					IF nCodingAndTrackingMode = 11 THEN
						FOR nPackIndex := 1 TO nMaxPackItem DO
							A_PackContentGenerator();
						END_FOR
					END_IF
	
					A_OuterEndPartGenerator();
					nOuterHeadCounter	:=nOuterHeadCounter +1;

				END_IF
	
			E_CS_ENDING:
				A_CaseEndPartGenerator();
				nCaseEndCounter :=	nCaseEndCounter	+1;
		END_CASE

		eState := E_XML_WRITEXML;
		nImigeProcessingSize	:= nImageByte;

	(* write XML file *)
	E_XML_WRITEXML:

		(* write XML image to file *)
		fbAppWriteFile(
			bExecute	:= TRUE,
			pSourceAddr	:= ADR(aXMLImage),
			nSourceSize	:= nImageByte,
			strPathFile	:= CONCAT(sPath, sFileName),
			tTimeout	:= T#3s,
		);

		(* file write complete *)
		IF fbAppWriteFile.bDone = TRUE THEN

			stWriteCHMFileStatistic.nTotalFilesWritten := stWriteCHMFileStatistic.nTotalFilesWritten + 1;

			(* file write completed OK *)
			IF fbAppWriteFile.bError = FALSE THEN

				(* correct no of bytes written to file *)
				IF fbAppWriteFile.nBytesWritten = nImageByte THEN

					stWriteCHMFileStatistic.nGoodFilesWritten := stWriteCHMFileStatistic.nGoodFilesWritten + 1;

					IF bCheckFileSize THEN
						eState := E_XML_CHECKFILESIZE;
					ELSE
						eState := E_XML_DONE;
					END_IF

				(* incorrect no of bytes written to file *)
				ELSE
					stWriteCHMFileStatistic.nBadFilesWritten :=stWriteCHMFileStatistic. nBadFilesWritten + 1;
				END_IF

			(* file write error *)
			ELSE

				bError := TRUE;
				nErrorID := fbAppWriteFile.nErrorID;
				eErrorState := eState;
				stWriteCHMFileStatistic.nFileWriteErrors := stWriteCHMFileStatistic.nFileWriteErrors + 1;

				eState := E_XML_DONE;
			END_IF

			(* close of fbWriteFile *)
			fbAppWriteFile(bExecute := FALSE);
		END_IF


	(* check XML file size is correct *)
	E_XML_CHECKFILESIZE:

		(* read XML file attributes *)
		fbGetFileInfo(
			bExecute		:= TRUE,
			strPathSource	:= sPath,
			strFileName	:= sFileName,
			tTimeout		:= T#1s,
		);

		(* read file attributes complete *)
		IF fbGetFileInfo.bDone = TRUE THEN

			stWriteCHMFileStatistic.nTotalFilesVerified := stWriteCHMFileStatistic.nTotalFilesVerified + 1;

			(* read file attributes completed OK *)
			IF fbGetFileInfo.bError = FALSE THEN

				(* file exists and file size is correct *)
				IF fbGetFileInfo.bFileExists = TRUE THEN

					(* file size is 0 bytes *)
					IF fbGetFileInfo.nFileSizeLo = 0 THEN

						stWriteCHMFileStatistic.nEmptyFilesVerified := stWriteCHMFileStatistic.nEmptyFilesVerified + 1;

					(* file size is not expected size *)
					ELSIF fbGetFileInfo.nFileSizeLo <> nImageByte THEN

						stWriteCHMFileStatistic.nSizeErrorsVerified :=stWriteCHMFileStatistic. nSizeErrorsVerified + 1;

					(* file size is correct *)
					ELSE

						stWriteCHMFileStatistic.nGoodFilesVerified := stWriteCHMFileStatistic.nGoodFilesVerified + 1;
					END_IF

					eState := E_XML_DONE;

				(* file not found *)
				ELSE

					bVerifyError := TRUE;
					stWriteCHMFileStatistic.nFileVerifyNotFound :=stWriteCHMFileStatistic.nFileVerifyNotFound + 1;

					IF bError = FALSE THEN

						bError := TRUE;
						nErrorID := 999;
						eErrorState := eState;
					END_IF

					eState := E_XML_DONE;
				END_IF

			(* read file attributes error *)
			ELSE

				stWriteCHMFileStatistic.nFileVerifyErrors := stWriteCHMFileStatistic.nFileVerifyErrors + 1;

				IF bError = FALSE THEN

					bError := TRUE;
					nErrorID := fbGetFileInfo.nErrorID;
					eErrorState := eState;
				END_IF

				eState := E_XML_DONE;
			END_IF

			(* close off fbFileSize *)
			fbGetFileInfo(bExecute := FALSE);
		END_IF


	(* sequence complete *)
	E_XML_DONE:

		(* update outputs *)
		bBusy := FALSE;
		bDone := TRUE;

		eState := E_XML_IDLE;
END_CASE

ACTION A_CaseEndPartGenerator:
	IF nCodingAndTrackingMode >= 7 THEN


				(* ItemList end*)
				sString := '$T$T$T$T</ItemList>$R$N';
				MEMMOVE(ADR(aXMLImage[nImageByte]), ADR(sString), LEN(sString));
				nImageByte := nImageByte + LEN(sString);

(***********CASE CONTENT END***********)
			(* Case Content END *)
			sString := '$T$T$T</Content>$R$N';
			MEMMOVE(ADR(aXMLImage[nImageByte]), ADR(sString), LEN(sString));
			nImageByte := nImageByte + LEN(sString);

	END_IF
			(* ProductionOrder *)
			sString := F_CONCAT3('$T$T$T<ProductionOrder>',stAgregationData.GenericHierarchy.CaseItem.ProductionOrder, '</ProductionOrder>$R$N');
			MEMMOVE(ADR(aXMLImage[nImageByte]), ADR(sString), LEN(sString));
			nImageByte := nImageByte + LEN(sString);

			(* LocalProductionOrder *)
			sString := F_CONCAT3('$T$T$T<LocalProductionOrder>',stAgregationData.GenericHierarchy.CaseItem.LocalProductionOrder, '</LocalProductionOrder>$R$N');
			MEMMOVE(ADR(aXMLImage[nImageByte]), ADR(sString), LEN(sString));
			nImageByte := nImageByte + LEN(sString);

			(* PITCode *)
			sString := F_CONCAT3('$T$T$T<PITCode>',stAgregationData.GenericHierarchy.CaseItem.PITCode, '</PITCode>$R$N');
			MEMMOVE(ADR(aXMLImage[nImageByte]), ADR(sString), LEN(sString));
			nImageByte := nImageByte + LEN(sString);

			(* BatchID *)
			sString := F_CONCAT3('$T$T$T<BatchID>',stAgregationData.GenericHierarchy.CaseItem.BatchID, '</BatchID>$R$N');
			MEMMOVE(ADR(aXMLImage[nImageByte]), ADR(sString), LEN(sString));
			nImageByte := nImageByte + LEN(sString);

			(* ProductionLine *)
			sString := F_CONCAT3('$T$T$T<ProductionLine>',stAgregationData.GenericHierarchy.CaseItem.ProductionLine, '</ProductionLine>$R$N');
			MEMMOVE(ADR(aXMLImage[nImageByte]), ADR(sString), LEN(sString));
			nImageByte := nImageByte + LEN(sString);


(***********Item CONTENT END***********)
		(* Item END *)
		sString := '$T$T</Item>$R$N';
		MEMMOVE(ADR(aXMLImage[nImageByte]), ADR(sString), LEN(sString));
		nImageByte := nImageByte + LEN(sString);

(***********GENERIC HIERARCHY CONTENT END***********)

	(* GenericHierarchy END *)
	sString := '$T</GenericHierarchy>$R$N';
	MEMMOVE(ADR(aXMLImage[nImageByte]), ADR(sString), LEN(sString));
	nImageByte := nImageByte + LEN(sString);

	(* Attributes *)
	sString := F_CONCAT3('$T<Attributes>', stAgregationData.Attributes.CSProductionTime, '</Attributes>$R$N');
	MEMMOVE(ADR(aXMLImage[nImageByte]), ADR(sString), LEN(sString));
	nImageByte := nImageByte + LEN(sString);

(* XPath leading tag  END*)
sString := '</GenericHierarchyList> $R$N';
MEMMOVE(ADR(aXMLImage[nImageByte]), ADR(sString), LEN(sString));
nImageByte := nImageByte + LEN(sString);
END_ACTION

ACTION A_CaseHeaderGenerator:
(* XML file version *)
(*sString := '<?xml version="1.0" encoding="utf-8"?>$R$N';
MEMMOVE(ADR(aXMLImage[nImageByte]), ADR(sString), LEN(sString));
nImageByte := nImageByte + LEN(sString);*)

(* XPath leading tag *)
sString := '<GenericHierarchyList xmlns:xsd="http://www.w3.org/2001/XMLSchema" xmlns:xsi="http://www.w3.org/2001/XMLSchema-instance"> $R$N';
MEMMOVE(ADR(aXMLImage[nImageByte]), ADR(sString), LEN(sString));
nImageByte := nImageByte + LEN(sString);

	(* MessageHeader *)
	sString := '$T<MessageHeader>$R$N';
	MEMMOVE(ADR(aXMLImage[nImageByte]), ADR(sString), LEN(sString));
	nImageByte := nImageByte + LEN(sString);

(***********MESSAGE HEADER CONTENT***********)

		(*(* CreationDate *)
		sString := F_CONCAT3('$T$T<CreationDate>',stAgregationData.MessageHeader.CreationDate, '</CreationDate>$R$N');
		MEMMOVE(ADR(aXMLImage[nImageByte]), ADR(sString), LEN(sString));
		nImageByte := nImageByte + LEN(sString);
	
		(* CreationTime *)
		sString := F_CONCAT3('$T$T<CreationTime>',stAgregationData.MessageHeader.CreationTime, '</CreationTime>$R$N');
		MEMMOVE(ADR(aXMLImage[nImageByte]), ADR(sString), LEN(sString));
		nImageByte := nImageByte + LEN(sString);*)

		(* ReferenceID *)
		sString := F_CONCAT3('$T$T<ReferenceID>',stAgregationData.MessageHeader.ReferenceID, '</ReferenceID>$R$N');
		MEMMOVE(ADR(aXMLImage[nImageByte]), ADR(sString), LEN(sString));
		nImageByte := nImageByte + LEN(sString);

		(* CreationTimeLocalUTC *)
		sString := F_CONCAT3('$T$T<CreationTimeLocalUTC>',stAgregationData.MessageHeader.CreationTimeLocalUTC, '</CreationTimeLocalUTC>$R$N');
		MEMMOVE(ADR(aXMLImage[nImageByte]), ADR(sString), LEN(sString));
		nImageByte := nImageByte + LEN(sString);

		(* MessageType *)
		sString := F_CONCAT3('$T$T<MessageType>',stAgregationData.MessageHeader.MessageType, '</MessageType>$R$N');
		MEMMOVE(ADR(aXMLImage[nImageByte]), ADR(sString), LEN(sString));
		nImageByte := nImageByte + LEN(sString);

		(* SenderSystem *)
		sString := F_CONCAT3('$T$T<SenderSystem>',stAgregationData.MessageHeader.SenderSystem, '</SenderSystem>$R$N');
		MEMMOVE(ADR(aXMLImage[nImageByte]), ADR(sString), LEN(sString));
		nImageByte := nImageByte + LEN(sString);

		(* ReceiverSystem *)
		sString := F_CONCAT3('$T$T<ReceiverSystem>',stAgregationData.MessageHeader.ReceiverSystem, '</ReceiverSystem>$R$N');
		MEMMOVE(ADR(aXMLImage[nImageByte]), ADR(sString), LEN(sString));
		nImageByte := nImageByte + LEN(sString);

(***********MESSAGE HEADER CONTENT END***********)

	(* MessageHeader END *)
	sString := '$T</MessageHeader>$R$N';
	MEMMOVE(ADR(aXMLImage[nImageByte]), ADR(sString), LEN(sString));
	nImageByte := nImageByte + LEN(sString);

	(* Factory*)
	sString := F_CONCAT3('$T<Factory>', stAgregationData.Factory, '</Factory>$R$N');
	MEMMOVE(ADR(aXMLImage[nImageByte]), ADR(sString), LEN(sString));
	nImageByte := nImageByte + LEN(sString);

	(* GenericHierarchy *)
	sString := '$T<GenericHierarchy>$R$N';
	MEMMOVE(ADR(aXMLImage[nImageByte]), ADR(sString), LEN(sString));
	nImageByte := nImageByte + LEN(sString);

(***********GENERIC HIERARCHY CONTENT***********)

		(* HierarchyType *)
		sString := F_CONCAT3('$T$T<HierarchyType>',stAgregationData.GenericHierarchy.HierarchyType, '</HierarchyType>$R$N');
		MEMMOVE(ADR(aXMLImage[nImageByte]), ADR(sString), LEN(sString));
		nImageByte := nImageByte + LEN(sString);

		(* PerformedAction *)
		sString := F_CONCAT3('$T$T<ACTION>',stAgregationData.GenericHierarchy.PerformedAction, '</ACTION>$R$N');
		MEMMOVE(ADR(aXMLImage[nImageByte]), ADR(sString), LEN(sString));
		nImageByte := nImageByte + LEN(sString);

		(* TrackingLevels *)
		sString := F_CONCAT3('$T$T<TrackingLevels>',stAgregationData.GenericHierarchy.TrackingLevels, '</TrackingLevels>$R$N');
		MEMMOVE(ADR(aXMLImage[nImageByte]), ADR(sString), LEN(sString));
		nImageByte := nImageByte + LEN(sString);

		(* TrackingIndicator *)
		sString := F_CONCAT3('$T$T<TrackingIndicator>',stAgregationData.GenericHierarchy.TrackingIndicator, '</TrackingIndicator>$R$N');
		MEMMOVE(ADR(aXMLImage[nImageByte]), ADR(sString), LEN(sString));
		nImageByte := nImageByte + LEN(sString);

		(* Item Type *)
		sString := '$T$T<Item Type="CS">$R$N';
		MEMMOVE(ADR(aXMLImage[nImageByte]), ADR(sString), LEN(sString));
		nImageByte := nImageByte + LEN(sString);

(***********Item Type CONTENT***********)
			(* Identity*)
			sString := '$T$T$T<Identity>$R$N';
			MEMMOVE(ADR(aXMLImage[nImageByte]), ADR(sString), LEN(sString));
			nImageByte := nImageByte + LEN(sString);

(***********Identity CONTENT***********)
					(* SKU *)
					sString := F_CONCAT3('$T$T$T$T<SKU>',stAgregationData.GenericHierarchy.CaseItem.Identity.SKU, '</SKU>$R$N');
					MEMMOVE(ADR(aXMLImage[nImageByte]), ADR(sString), LEN(sString));
					nImageByte := nImageByte + LEN(sString);

					(* GTIN *)
					sString := F_CONCAT3('$T$T$T$T<GTIN>',stAgregationData.GenericHierarchy.CaseItem.Identity.GTIN, '</GTIN>$R$N');
					MEMMOVE(ADR(aXMLImage[nImageByte]), ADR(sString), LEN(sString));
					nImageByte := nImageByte + LEN(sString);

					(* ID *)
					sString := F_CONCAT3('$T$T$T$T<ID>',stAgregationData.GenericHierarchy.CaseItem.Identity.ID, '</ID>$R$N');
					MEMMOVE(ADR(aXMLImage[nImageByte]), ADR(sString), LEN(sString));
					nImageByte := nImageByte + LEN(sString);

					(* ReadQuality *)
					sString := F_CONCAT3('$T$T$T$T<ReadQuality>',stAgregationData.GenericHierarchy.CaseItem.Identity.ReadQuality, '</ReadQuality>$R$N');
					MEMMOVE(ADR(aXMLImage[nImageByte]), ADR(sString), LEN(sString));
					nImageByte := nImageByte + LEN(sString);

(***********Identity CONTENT END***********)

			(* Identity END *)
			sString := '$T$T$T</Identity>$R$N';
			MEMMOVE(ADR(aXMLImage[nImageByte]), ADR(sString), LEN(sString));
			nImageByte := nImageByte + LEN(sString);

			(* ItemState *)
			sString := F_CONCAT3('$T$T$T<ItemState>',stAgregationData.GenericHierarchy.CaseItem.ItemState, '</ItemState>$R$N');
			MEMMOVE(ADR(aXMLImage[nImageByte]), ADR(sString), LEN(sString));
			nImageByte := nImageByte + LEN(sString);

			(* RejectReason *)
			sString := '$T$T$T<RejectReason>$R$N';
			MEMMOVE(ADR(aXMLImage[nImageByte]), ADR(sString), LEN(sString));
			nImageByte := nImageByte + LEN(sString);

				sString := F_CONCAT3('$T$T$T$T<Reason>',stAgregationData.GenericHierarchy.CaseItem.RejectReason, '</Reason>$R$N');
				MEMMOVE(ADR(aXMLImage[nImageByte]), ADR(sString), LEN(sString));
				nImageByte := nImageByte + LEN(sString);

			sString := '$T$T$T</RejectReason>$R$N';
			MEMMOVE(ADR(aXMLImage[nImageByte]), ADR(sString), LEN(sString));
			nImageByte := nImageByte + LEN(sString);

			(*logs *)
			sString := '$T$T$T<logs>$R$N';
			MEMMOVE(ADR(aXMLImage[nImageByte]), ADR(sString), LEN(sString));
			nImageByte := nImageByte + LEN(sString);

				(* TimeStamp *)
				sString := F_CONCAT3('$T$T$T$T<TimeStamp Topic="Aggregation">',stAgregationData.GenericHierarchy.CaseItem.TimeStamp, '</TimeStamp>$R$N');
				MEMMOVE(ADR(aXMLImage[nImageByte]), ADR(sString), LEN(sString));
				nImageByte := nImageByte + LEN(sString);

			(* logs END *)
			sString := '$T$T$T</logs>$R$N';
			MEMMOVE(ADR(aXMLImage[nImageByte]), ADR(sString), LEN(sString));
			nImageByte := nImageByte + LEN(sString);

			(* NoRead *)
			sString := F_CONCAT3('$T$T$T<NoRead>',stAgregationData.GenericHierarchy.CaseItem.NoRead, '</NoRead>$R$N');
			MEMMOVE(ADR(aXMLImage[nImageByte]), ADR(sString), LEN(sString));
			nImageByte := nImageByte + LEN(sString);

(***********CONTENT***********)
	IF nCodingAndTrackingMode >= 7 THEN

			(* Case Content *)
			sString := '$T$T$T<Content>$R$N';
			MEMMOVE(ADR(aXMLImage[nImageByte]), ADR(sString), LEN(sString));
			nImageByte := nImageByte + LEN(sString);

				(* Case DefaultIdentity*)
				sString := '$T$T$T$T<DefaultIdentity>$R$N';
				MEMMOVE(ADR(aXMLImage[nImageByte]), ADR(sString), LEN(sString));
				nImageByte := nImageByte + LEN(sString);

						(* SKU *)
						sString := F_CONCAT3('$T$T$T$T$T<SKU>',stAgregationData.GenericHierarchy.CaseItem.Content.DefaultIdentity.SKU, '</SKU>$R$N');
						MEMMOVE(ADR(aXMLImage[nImageByte]), ADR(sString), LEN(sString));
						nImageByte := nImageByte + LEN(sString);

						(* GTIN *)
						sString := F_CONCAT3('$T$T$T$T$T<GTIN>',stAgregationData.GenericHierarchy.CaseItem.Content.DefaultIdentity.GTIN, '</GTIN>$R$N');
						MEMMOVE(ADR(aXMLImage[nImageByte]), ADR(sString), LEN(sString));
						nImageByte := nImageByte + LEN(sString);

						(* ProductionOrder *)
						sString := F_CONCAT3('$T$T$T$T$T<ProductionOrder>',stAgregationData.GenericHierarchy.CaseItem.Content.DefaultIdentity.ProductionOrder, '</ProductionOrder>$R$N');
						MEMMOVE(ADR(aXMLImage[nImageByte]), ADR(sString), LEN(sString));
						nImageByte := nImageByte + LEN(sString);

						(* LocalProductionOrder *)
						sString := F_CONCAT3('$T$T$T$T$T<LocalProductionOrder>',stAgregationData.GenericHierarchy.CaseItem.Content.DefaultIdentity.LocalProductionOrder, '</LocalProductionOrder>$R$N');
						MEMMOVE(ADR(aXMLImage[nImageByte]), ADR(sString), LEN(sString));
						nImageByte := nImageByte + LEN(sString);

						(* PITCode *)
						sString := F_CONCAT3('$T$T$T$T$T<PITCode>',stAgregationData.GenericHierarchy.CaseItem.Content.DefaultIdentity.PITCode, '</PITCode>$R$N');
						MEMMOVE(ADR(aXMLImage[nImageByte]), ADR(sString), LEN(sString));
						nImageByte := nImageByte + LEN(sString);

						(* BatchID *)
						sString := F_CONCAT3('$T$T$T$T$T<BatchID>',stAgregationData.GenericHierarchy.CaseItem.Content.DefaultIdentity.BatchID, '</BatchID>$R$N');
						MEMMOVE(ADR(aXMLImage[nImageByte]), ADR(sString), LEN(sString));
						nImageByte := nImageByte + LEN(sString);

						(* ProductionLine *)
						sString := F_CONCAT3('$T$T$T$T$T<ProductionLine>',stAgregationData.GenericHierarchy.CaseItem.Content.DefaultIdentity.ProductionLine, '</ProductionLine>$R$N');
						MEMMOVE(ADR(aXMLImage[nImageByte]), ADR(sString), LEN(sString));
						nImageByte := nImageByte + LEN(sString);

				(* Case DefaultIdentity END*)
				sString := '$T$T$T$T</DefaultIdentity>$R$N';
				MEMMOVE(ADR(aXMLImage[nImageByte]), ADR(sString), LEN(sString));
				nImageByte := nImageByte + LEN(sString);

				(* ExpectedItemCount *)
				sString := F_CONCAT3('$T$T$T$T<ExpectedItemCount>',stAgregationData.GenericHierarchy.CaseItem.Content.ExpectedItemCount, '</ExpectedItemCount>$R$N');
				MEMMOVE(ADR(aXMLImage[nImageByte]), ADR(sString), LEN(sString));
				nImageByte := nImageByte + LEN(sString);

				(* ItemReadRate *)
				sString := F_CONCAT3('$T$T$T$T<ItemReadRate>',stAgregationData.GenericHierarchy.CaseItem.Content.ItemReadRate, '</ItemReadRate>$R$N');
				MEMMOVE(ADR(aXMLImage[nImageByte]), ADR(sString), LEN(sString));
				nImageByte := nImageByte + LEN(sString);

				(* ItemList*)
				sString := '$T$T$T$T<ItemList>$R$N';
				MEMMOVE(ADR(aXMLImage[nImageByte]), ADR(sString), LEN(sString));
				nImageByte := nImageByte + LEN(sString);
	END_IF
END_ACTION

ACTION A_OuterEndPartGenerator:
(*
    </ItemList> 
                        </Content> 
                    </Item> 

*)
						IF nCodingAndTrackingMode = 11 THEN
								(* ItemList end*)
								sString := '$T$T$T$T$T$T$T</ItemList>$R$N';
								MEMMOVE(ADR(aXMLImage[nImageByte]), ADR(sString), LEN(sString));
								nImageByte := nImageByte + LEN(sString);
	(***********CASE CONTENT END***********)
							(* Outer Content END *)
							sString := '$T$T$T$T$T$T</Content>$R$N';
							MEMMOVE(ADR(aXMLImage[nImageByte]), ADR(sString), LEN(sString));
							nImageByte := nImageByte + LEN(sString);
						END_IF

								(* Item Type END *)
								sString := '$T$T$T$T$T</Item>$R$N';
							MEMMOVE(ADR(aXMLImage[nImageByte]), ADR(sString), LEN(sString));
							nImageByte := nImageByte + LEN(sString);
END_ACTION

ACTION A_OuterHeaderContentGenerator:
(*
                  <Item Type="OUT"> 
                        <Identity> 
                         	   <ID>55128CY203644964300</ID> 
                        	    <ReadQuality>100</ReadQuality> 
                        </Identity> 
                        <ItemState>Verified</ItemState> 
                        <RejectReason /> 
                        <logs> 
                   		        <TimeStamp Topic="Aggregation">2018-03-22T20:46:01.5229666+01:00</TimeStamp> 
                        </logs> 
                        <NoRead>false</NoRead> 
                        <Content> 
                           	 <DefaultIdentity> 
                      	     	     <SKU>10045622</SKU> 
                        	   	     <GTIN>00000087295993</GTIN> 
                        		        <ProductionOrder>2523549</ProductionOrder> 
                         		       <LocalProductionOrder>2523549</LocalProductionOrder> 
                           		     <PITCode>3</PITCode> 
                          		      <BatchID>55122018</BatchID> 
                        		        <ProductionLine>12</ProductionLine> 
                       	     </DefaultIdentity> 
                      	      <ExpectedItemCount>10</ExpectedItemCount> 
                       	     <ItemReadRate>100</ItemReadRate> 
                       	     <ItemList> 

*)


					(* Item Type *)
					sString := '$T$T$T$T$T<Item Type="OUT">$R$N';
					MEMMOVE(ADR(aXMLImage[nImageByte]), ADR(sString), LEN(sString));
					nImageByte := nImageByte + LEN(sString);

						(* Identity *)
						sString := '$T$T$T$T$T$T<Identity>$R$N';
						MEMMOVE(ADR(aXMLImage[nImageByte]), ADR(sString), LEN(sString));
						nImageByte := nImageByte + LEN(sString);

							(* ID *)
							sString := F_CONCAT3('$T$T$T$T$T$T$T<ID><![CDATA[',stAgregationData.GenericHierarchy.CaseItem.Content.arrOuterItem[nOuterIndex].Identity.ID, ']]></ID>$R$N');
							MEMMOVE(ADR(aXMLImage[nImageByte]), ADR(sString), LEN(sString));
							nImageByte := nImageByte + LEN(sString);

							(* ReadQuality *)
							sString := F_CONCAT3('$T$T$T$T$T$T$T<ReadQuality>',stAgregationData.GenericHierarchy.CaseItem.Content.arrOuterItem[nOuterIndex].Identity.ReadQuality, '</ReadQuality>$R$N');
							MEMMOVE(ADR(aXMLImage[nImageByte]), ADR(sString), LEN(sString));
							nImageByte := nImageByte + LEN(sString);

						(* Identity END *)
						sString := '$T$T$T$T$T$T</Identity>$R$N';
						MEMMOVE(ADR(aXMLImage[nImageByte]), ADR(sString), LEN(sString));
						nImageByte := nImageByte + LEN(sString);


						(* ItemState *)
						sString := F_CONCAT3('$T$T$T$T$T$T<ItemState>',stAgregationData.GenericHierarchy.CaseItem.Content.arrOuterItem[nOuterIndex].ItemState, '</ItemState>$R$N');
						MEMMOVE(ADR(aXMLImage[nImageByte]), ADR(sString), LEN(sString));
						nImageByte := nImageByte + LEN(sString);

						(* RejectReason *)
						sString := '$T$T$T$T$T$T<RejectReason>$R$N';
						MEMMOVE(ADR(aXMLImage[nImageByte]), ADR(sString), LEN(sString));
						nImageByte := nImageByte + LEN(sString);
			
							sString := F_CONCAT3('$T$T$T$T$T$T$T<Reason>',stAgregationData.GenericHierarchy.CaseItem.Content.arrOuterItem[nOuterIndex].RejectReason, '</Reason>$R$N');
							MEMMOVE(ADR(aXMLImage[nImageByte]), ADR(sString), LEN(sString));
							nImageByte := nImageByte + LEN(sString);
			
						sString := '$T$T$T$T$T$T</RejectReason>$R$N';
						MEMMOVE(ADR(aXMLImage[nImageByte]), ADR(sString), LEN(sString));
						nImageByte := nImageByte + LEN(sString);


						(*logs *)
						sString := '$T$T$T$T$T$T<logs>$R$N';
						MEMMOVE(ADR(aXMLImage[nImageByte]), ADR(sString), LEN(sString));
						nImageByte := nImageByte + LEN(sString);

							(* TimeStamp *)
							sString := F_CONCAT3('$T$T$T$T$T$T$T<TimeStamp Topic="Aggregation">',stAgregationData.GenericHierarchy.CaseItem.Content.arrOuterItem[nOuterIndex].TimeStamp, '</TimeStamp>$R$N');
							MEMMOVE(ADR(aXMLImage[nImageByte]), ADR(sString), LEN(sString));
							nImageByte := nImageByte + LEN(sString);

						(* logs END *)
						sString := '$T$T$T$T$T$T</logs>$R$N';
						MEMMOVE(ADR(aXMLImage[nImageByte]), ADR(sString), LEN(sString));
						nImageByte := nImageByte + LEN(sString);

						(* NoRead *)
						sString := F_CONCAT3('$T$T$T$T$T$T<NoRead>',stAgregationData.GenericHierarchy.CaseItem.Content.arrOuterItem[nOuterIndex].NoRead, '</NoRead>$R$N');
						MEMMOVE(ADR(aXMLImage[nImageByte]), ADR(sString), LEN(sString));
						nImageByte := nImageByte + LEN(sString);
(***********CONTENT***********)

						IF nCodingAndTrackingMode = 11 THEN
							(* Outer Content *)
							sString := '$T$T$T$T$T$T<Content>$R$N';
							MEMMOVE(ADR(aXMLImage[nImageByte]), ADR(sString), LEN(sString));
							nImageByte := nImageByte + LEN(sString);
	
	
								(* Case DefaultIdentity*)
								sString := '$T$T$T$T$T$T$T<DefaultIdentity>$R$N';
								MEMMOVE(ADR(aXMLImage[nImageByte]), ADR(sString), LEN(sString));
								nImageByte := nImageByte + LEN(sString);
	
										(* SKU *)
										sString := F_CONCAT3('$T$T$T$T$T$T$T$T<SKU>',stAgregationData.GenericHierarchy.CaseItem.Content.arrOuterItem[nOuterIndex].Content.DefaultIdentity.SKU, '</SKU>$R$N');
										MEMMOVE(ADR(aXMLImage[nImageByte]), ADR(sString), LEN(sString));
										nImageByte := nImageByte + LEN(sString);
	
										(* GTIN *)
										sString := F_CONCAT3('$T$T$T$T$T$T$T$T<GTIN>',stAgregationData.GenericHierarchy.CaseItem.Content.arrOuterItem[nOuterIndex].Content.DefaultIdentity.GTIN, '</GTIN>$R$N');
										MEMMOVE(ADR(aXMLImage[nImageByte]), ADR(sString), LEN(sString));
										nImageByte := nImageByte + LEN(sString);
	
										(* ProductionOrder *)
										sString := F_CONCAT3('$T$T$T$T$T$T$T$T<ProductionOrder>',stAgregationData.GenericHierarchy.CaseItem.Content.arrOuterItem[nOuterIndex].Content.DefaultIdentity.ProductionOrder, '</ProductionOrder>$R$N');
										MEMMOVE(ADR(aXMLImage[nImageByte]), ADR(sString), LEN(sString));
										nImageByte := nImageByte + LEN(sString);
	
										(* LocalProductionOrder *)
										sString := F_CONCAT3('$T$T$T$T$T$T$T$T<LocalProductionOrder>',stAgregationData.GenericHierarchy.CaseItem.Content.arrOuterItem[nOuterIndex].Content.DefaultIdentity.LocalProductionOrder, '</LocalProductionOrder>$R$N');
										MEMMOVE(ADR(aXMLImage[nImageByte]), ADR(sString), LEN(sString));
										nImageByte := nImageByte + LEN(sString);
	
										(* PITCode *)
										sString := F_CONCAT3('$T$T$T$T$T$T$T$T<PITCode>',stAgregationData.GenericHierarchy.CaseItem.Content.arrOuterItem[nOuterIndex].Content.DefaultIdentity.PITCode, '</PITCode>$R$N');
										MEMMOVE(ADR(aXMLImage[nImageByte]), ADR(sString), LEN(sString));
										nImageByte := nImageByte + LEN(sString);
	
										(* BatchID *)
										sString := F_CONCAT3('$T$T$T$T$T$T$T$T<BatchID>',stAgregationData.GenericHierarchy.CaseItem.Content.arrOuterItem[nOuterIndex].Content.DefaultIdentity.BatchID, '</BatchID>$R$N');
										MEMMOVE(ADR(aXMLImage[nImageByte]), ADR(sString), LEN(sString));
										nImageByte := nImageByte + LEN(sString);
	
										(* ProductionLine *)
										sString := F_CONCAT3('$T$T$T$T$T$T$T$T<ProductionLine>',stAgregationData.GenericHierarchy.CaseItem.Content.arrOuterItem[nOuterIndex].Content.DefaultIdentity.ProductionLine, '</ProductionLine>$R$N');
										MEMMOVE(ADR(aXMLImage[nImageByte]), ADR(sString), LEN(sString));
										nImageByte := nImageByte + LEN(sString);
	
								(* Case DefaultIdentity END*)
								sString := '$T$T$T$T$T$T$T</DefaultIdentity>$R$N';
								MEMMOVE(ADR(aXMLImage[nImageByte]), ADR(sString), LEN(sString));
								nImageByte := nImageByte + LEN(sString);
	
								(* ExpectedItemCount *)
								sString := F_CONCAT3('$T$T$T$T$T$T$T<ExpectedItemCount>',stAgregationData.GenericHierarchy.CaseItem.Content.arrOuterItem[nOuterIndex].Content.ExpectedItemCount, '</ExpectedItemCount>$R$N');
								MEMMOVE(ADR(aXMLImage[nImageByte]), ADR(sString), LEN(sString));
								nImageByte := nImageByte + LEN(sString);
	
								(* ItemReadRate *)
								sString := F_CONCAT3('$T$T$T$T$T$T$T<ItemReadRate>',stAgregationData.GenericHierarchy.CaseItem.Content.arrOuterItem[nOuterIndex].Content.ItemReadRate, '</ItemReadRate>$R$N');
								MEMMOVE(ADR(aXMLImage[nImageByte]), ADR(sString), LEN(sString));
								nImageByte := nImageByte + LEN(sString);
	
								(* ItemList*)
								sString := '$T$T$T$T$T$T$T<ItemList>$R$N';
								MEMMOVE(ADR(aXMLImage[nImageByte]), ADR(sString), LEN(sString));
								nImageByte := nImageByte + LEN(sString);
						END_IF
END_ACTION

ACTION A_PackContentGenerator:
(*
                             <Item Type="PK"> 
                                    <Identity> 
                                        <ID>1XJWVXUS1FM7</ID> 
                                        <ReadQuality>100</ReadQuality> 
                                    </Identity> 
                                    <ItemState>Verified</ItemState> 
                                    <RejectReason /> 
                                    <logs> 
                                        <TimeStamp Topic="Aggregation">2018-03-22T20:45:38.4129952+01:00</TimeStamp> 
                                    </logs> 
                                    <NoRead>false</NoRead> 
                                </Item> 
*)

								(* Item Type *)
								sString := '$T$T$T$T$T$T$T$T<Item Type="PK">$R$N';
								MEMMOVE(ADR(aXMLImage[nImageByte]), ADR(sString), LEN(sString));
								nImageByte := nImageByte + LEN(sString);

									(* Identity *)
									sString := '$T$T$T$T$T$T$T$T$T<Identity>$R$N';
									MEMMOVE(ADR(aXMLImage[nImageByte]), ADR(sString), LEN(sString));
									nImageByte := nImageByte + LEN(sString);

										(* ID *)
										sString := F_CONCAT3('$T$T$T$T$T$T$T$T$T$T<ID><![CDATA[',stAgregationData.GenericHierarchy.CaseItem.Content.arrOuterItem[nOuterIndex].Content.arrPackItem[nPackIndex].Identity.ID, ']]></ID>$R$N');
										MEMMOVE(ADR(aXMLImage[nImageByte]), ADR(sString), LEN(sString));
										nImageByte := nImageByte + LEN(sString);

										(* ReadQuality *)
										sString := F_CONCAT3('$T$T$T$T$T$T$T$T$T$T<ReadQuality>',stAgregationData.GenericHierarchy.CaseItem.Content.arrOuterItem[nOuterIndex].Content.arrPackItem[nPackIndex].Identity.ReadQuality, '</ReadQuality>$R$N');
										MEMMOVE(ADR(aXMLImage[nImageByte]), ADR(sString), LEN(sString));
										nImageByte := nImageByte + LEN(sString);

									(* Identity END *)
									sString := '$T$T$T$T$T$T$T$T$T</Identity>$R$N';
									MEMMOVE(ADR(aXMLImage[nImageByte]), ADR(sString), LEN(sString));
									nImageByte := nImageByte + LEN(sString);

									(* ItemState *)
									sString := F_CONCAT3('$T$T$T$T$T$T$T$T$T<ItemState>',stAgregationData.GenericHierarchy.CaseItem.Content.arrOuterItem[nOuterIndex].Content.arrPackItem[nPackIndex].ItemState, '</ItemState>$R$N');
									MEMMOVE(ADR(aXMLImage[nImageByte]), ADR(sString), LEN(sString));
									nImageByte := nImageByte + LEN(sString);
			

									(* RejectReason *)
									sString := '$T$T$T$T$T$T$T$T$T<RejectReason>$R$N';
									MEMMOVE(ADR(aXMLImage[nImageByte]), ADR(sString), LEN(sString));
									nImageByte := nImageByte + LEN(sString);

										sString := F_CONCAT3('$T$T$T$T$T$T$T$T$T$T<Reason>',stAgregationData.GenericHierarchy.CaseItem.Content.arrOuterItem[nOuterIndex].Content.arrPackItem[nPackIndex].RejectReason, '</Reason>$R$N');
										MEMMOVE(ADR(aXMLImage[nImageByte]), ADR(sString), LEN(sString));
										nImageByte := nImageByte + LEN(sString);
			
									sString := '$T$T$T$T$T$T$T$T$T</RejectReason>$R$N';
									MEMMOVE(ADR(aXMLImage[nImageByte]), ADR(sString), LEN(sString));
									nImageByte := nImageByte + LEN(sString);


									(*logs *)
									sString := '$T$T$T$T$T$T$T$T$T<logs>$R$N';
									MEMMOVE(ADR(aXMLImage[nImageByte]), ADR(sString), LEN(sString));
									nImageByte := nImageByte + LEN(sString);
	
										(* TimeStamp *)
										sString := F_CONCAT3('$T$T$T$T$T$T$T$T$T$T<TimeStamp Topic="Aggregation">',stAgregationData.GenericHierarchy.CaseItem.Content.arrOuterItem[nOuterIndex].Content.arrPackItem[nPackIndex].TimeStamp, '</TimeStamp>$R$N');
										MEMMOVE(ADR(aXMLImage[nImageByte]), ADR(sString), LEN(sString));
										nImageByte := nImageByte + LEN(sString);
			
									(* logs END *)
									sString := '$T$T$T$T$T$T$T$T$T</logs>$R$N';
									MEMMOVE(ADR(aXMLImage[nImageByte]), ADR(sString), LEN(sString));
									nImageByte := nImageByte + LEN(sString);

									(* No Read *)
									sString := F_CONCAT3('$T$T$T$T$T$T$T$T$T<NoRead>',stAgregationData.GenericHierarchy.CaseItem.Content.arrOuterItem[nOuterIndex].Content.arrPackItem[nPackIndex].NoRead, '</NoRead>$R$N');
									MEMMOVE(ADR(aXMLImage[nImageByte]), ADR(sString), LEN(sString));
									nImageByte := nImageByte + LEN(sString);

								(* Item Type END *)
								sString := '$T$T$T$T$T$T$T$T</Item>$R$N';
								MEMMOVE(ADR(aXMLImage[nImageByte]), ADR(sString), LEN(sString));
								nImageByte := nImageByte + LEN(sString);
END_ACTION

END_FUNCTION_BLOCK

// ---- POUs/_Exclude/v1_1/FB_CHM_XMLImageGenerator.TcPOU
FUNCTION_BLOCK FB_CHM_XMLImageGenerator
VAR_INPUT
	bExecute						: BOOL;
	sLocalCHMPath				: STRING(50);
	sCHMFileName					: T_CHM_Filename;	(* current PCM file *)
	nMaxOuterItem				: UINT	:=50;
	nMaxPackItem					: UINT	:=10;
	bClearStatistic					: BOOL;
	nCodingAndTrackingMode		: INT;
	tTimeOut						: TIME;
	bIsValid						: BOOL;
END_VAR
VAR_IN_OUT
	stCHMDataStruct				: ST_CHM_Data;
END_VAR
VAR_OUTPUT
	bDone							: BOOL;					(* TRUE = XML file write complete *)
	bBusy							: BOOL;					(* TRUE = XML file write in progress *)
	bError							: BOOL;					(* TRUE = XML file write error *)
	nErrorID						: UDINT;				(* file write error code *)
	stLastCaseHierarchyMessage	: ST_CHM_Data;
	nLastImigeSize					: UDINT;
	tPerformanceRate				 :TIME;

END_VAR
VAR
	eXMLStep				: E_XML_GeneratorState;
	eErrorState				: E_XML_GeneratorState;

	rtrigExecute			:	R_TRIG;
	rtrigFBDone			:	R_TRIG;

	tonTimeOut			:	TON;
	tonPerfomance		:	TON;

	fbWriteCHMDataToXML	:	FB_CHM_BiuldXMLImige;
	fbCreateFLGFile		:	FB_CHM_SaveFLG_File;

	(*eXMLMode			:	E_XML_WritingMode;*)
	eCurrentXMLMode		: 	E_XML_WritingMode;

	aImigeSize			:	 ARRAY[0..100] OF UDINT;

	bWriteCaseDataToXML	:	BOOL;
	nCHMOuterIndex		: 	UINT := 1;
	nMaxCHMOuterIndex	: 	UINT;

	bCheckFileSize			: 	BOOL;
	bCreatFLGFileExe		: 	BOOL;

	nSequenceNumber		: 	INT;

END_VAR

rtrigExecute(CLK:=bExecute);

tonTimeOut(IN:= eXMLStep<>E_XML_GENERATOR_IDLE, PT:= tTimeOut);

IF tonTimeOut.Q AND tTimeOut <> t#0ms THEN

	bDone	:=  	TRUE;
	bBusy	:=  	FALSE;
	bError	:= 	TRUE;
	nErrorID	:= 	1;

	bWriteCaseDataToXML	:= FALSE;
	bCheckFileSize			:= FALSE;
	bCreatFLGFileExe		:= FALSE;

	tPerformanceRate := tonPerfomance.ET;

	eXMLStep	:=E_XML_GENERATOR_IDLE;
END_IF

tonPerfomance(IN:= eXMLStep<>E_XML_GENERATOR_IDLE, PT:= t#30s);

IF bClearStatistic THEN
	MEMSET(ADR(aImigeSize), 16#00, SIZEOF(aImigeSize));
END_IF

CASE eXMLStep OF

	E_XML_GENERATOR_IDLE:
	
		IF rtrigExecute.Q THEN

			(* update outputs *)
			bDone := FALSE;
			bBusy := TRUE;
			bError := FALSE;
			nErrorID := 0;
	
			eErrorState := eXMLStep;
	
			bWriteCaseDataToXML	:= FALSE;
			bCheckFileSize			:= FALSE;
			bCreatFLGFileExe		:= FALSE;
			nCHMOuterIndex		:= 1;

			MEMSET(ADR(stLastCaseHierarchyMessage), 16#00, SIZEOF(stLastCaseHierarchyMessage));
	
			nLastImigeSize		:= 0;
			tPerformanceRate		 :=t#0ms;

			eXMLStep	:=E_XML_GENERATE_HEAD_CHM;

		ELSIF	NOT bExecute THEN

			bDone 	:= FALSE;
			bBusy 	:= FALSE;
			(*bError 	:= FALSE;
			nErrorID	 := 0;*)
	
			bWriteCaseDataToXML	:= FALSE;
			bCheckFileSize			:= FALSE;
			bCreatFLGFileExe		:= FALSE;

		END_IF
	
	E_XML_GENERATE_HEAD_CHM:
	
		MEMSET(ADR(aImigeSize), 16#00, SIZEOF(aImigeSize));
	
		bWriteCaseDataToXML := TRUE;
		bCheckFileSize	:=	TRUE;
		eCurrentXMLMode := E_CS_HEADER;
	
		IF fbWriteCHMDataToXML.bBusy THEN
	
			eXMLStep	:=E_XML_DONE_HEAD_CHM;
		END_IF
	
	E_XML_DONE_HEAD_CHM:
	
		bWriteCaseDataToXML := FALSE;
	
	
		IF	fbWriteCHMDataToXML.bError	THEN
	
			bError 	:= TRUE;
			nErrorID	 := fbWriteCHMDataToXML.nErrorID;
			eErrorState := eXMLStep;
	
			eXMLStep	:=E_XML_GENERATOR_DONE;
	
		ELSIF fbWriteCHMDataToXML.bDone THEN
	
			eXMLStep	:=E_XML_GENERATE_BODY_CHM;
		END_IF

	E_XML_GENERATE_BODY_CHM:

		bCheckFileSize	:=	FALSE;
		bWriteCaseDataToXML := TRUE;
		eCurrentXMLMode := E_OUTER_HEADER;
	
		IF fbWriteCHMDataToXML.bBusy THEN
	
			eXMLStep	:=E_XML_DONE_BODY_CHM;
		END_IF
	
	E_XML_DONE_BODY_CHM:
	
		bWriteCaseDataToXML := FALSE;
	
		IF	fbWriteCHMDataToXML.bError	THEN

			bError 	:= TRUE;
			nErrorID	 := fbWriteCHMDataToXML.nErrorID;
			eErrorState := eXMLStep;
	
			eXMLStep	:=E_XML_GENERATOR_DONE;
	
		ELSIF fbWriteCHMDataToXML.bDone AND nCHMOuterIndex >= nMaxOuterItem  THEN
	
			eXMLStep	:=E_XML_GENERATE_ENDING_CHM;
	
		ELSIF fbWriteCHMDataToXML.bDone THEN

			nCHMOuterIndex	:=	nCHMOuterIndex+1;
	
			eXMLStep	:=E_XML_GENERATE_BODY_CHM;
		END_IF
	
	E_XML_GENERATE_ENDING_CHM:
	
		bWriteCaseDataToXML := TRUE;
		bCheckFileSize	:=	TRUE;
		eCurrentXMLMode := E_CS_ENDING;
	
		IF fbWriteCHMDataToXML.bBusy THEN
	
			eXMLStep	:=E_XML_DONE_ENDING_CHM;
		END_IF
	
	E_XML_DONE_ENDING_CHM:
	
		bWriteCaseDataToXML := FALSE;
	
		IF	fbWriteCHMDataToXML.bError	THEN

			bError 	:= TRUE;
			nErrorID	 := fbWriteCHMDataToXML.nErrorID;
			eErrorState := eXMLStep;
	
			eXMLStep	:=E_XML_GENERATOR_DONE;

		ELSIF fbWriteCHMDataToXML.bDone THEN

			nMaxCHMOuterIndex	:= nCHMOuterIndex;
			nCHMOuterIndex	:= 1;
			tPerformanceRate := tonPerfomance.ET;

			IF bIsValid THEN
				eXMLStep	:=E_XML_GENERATE_FLG;
			ELSE
				eXMLStep	:=E_XML_GENERATOR_DONE;
			END_IF
		END_IF

	E_XML_GENERATE_FLG:

		bCreatFLGFileExe := TRUE;
	
		IF fbCreateFLGFile.bBusy THEN
	
			eXMLStep	:=E_XML_DONE_FLG;
		END_IF
	
	E_XML_DONE_FLG:
	
		bCreatFLGFileExe := FALSE;
	
		IF	fbCreateFLGFile.bError	THEN

			bError 	:= TRUE;
			nErrorID	 := fbCreateFLGFile.nErrorID;
			eErrorState := eXMLStep;
	
			eXMLStep	:=E_XML_GENERATOR_DONE;
	
		ELSIF fbCreateFLGFile.bDone THEN
	
			nSequenceNumber	:= nSequenceNumber+1;
	
			eXMLStep	:=E_XML_GENERATOR_DONE;
		END_IF

	E_XML_GENERATOR_DONE:
	
		MEMCPY(ADR(stLastCaseHierarchyMessage), ADR(stCHMDataStruct), SIZEOF(stCHMDataStruct));

		bDone	:=  TRUE;
		bBusy	:=  FALSE;

		eXMLStep	:=E_XML_GENERATOR_IDLE;
	

ELSE

	eXMLStep	:=E_XML_GENERATOR_IDLE;
END_CASE

fbWriteCHMDataToXML(
	bExecute							:= bWriteCaseDataToXML,					(* set TRUE to write Case Produced file *)
	sPath							:= sLocalCHMPath,	(* path for target file C:\CaseTrace*)
	sFileName						:=sCHMFileName,
	stAgregationData					:=stCHMDataStruct,		(* case data to be written to XML *)
	stWriteCHMFileStatistic				:=stWriteCHMFileStatistic,
	eMode							:= eCurrentXMLMode,
	nMaxPackItem						:= nMaxPackItem,
	nOuterIndex						:=nCHMOuterIndex,
	bCheckFileSize						:=bCheckFileSize,
	nCodingAndTrackingMode			:=nCodingAndTrackingMode,
	bDone							=>,					(* TRUE = XML file write complete *)
	bBusy							=>,					(* TRUE = XML file write in progress *)
	bError							=> ,					(* TRUE = XML file write error *)
	nErrorID							=>,				(* file write error code *)
	bVerifyError						=>,				(* TRUE = XML file verification error *)
	nImigeProcessingSize				=>
);

rtrigFBDone(CLK:= fbWriteCHMDataToXML.bDone);

IF	rtrigFBDone.Q	THEN
	nLastImigeSize	:= fbWriteCHMDataToXML.nImigeProcessingSize;
	MEMMOVE(ADR(aImigeSize[1]), ADR(aImigeSize), SIZEOF(aImigeSize)-SIZEOF(aImigeSize[1]));
	aImigeSize[0] := nLastImigeSize;
END_IF

fbCreateFLGFile(
	bExecute							:= bCreatFLGFileExe,					(* set TRUE to write Case Produced file *)
	sPath							:= sLocalCHMPath,			(* path for target file C:\CaseTrace*)
	sFLGFileName						:=sCHMFileName,
	bDone							=>,					(* TRUE = XML file write complete *)
	bBusy							=>,					(* TRUE = XML file write in progress *)
	bError							=>,					(* TRUE = XML file write error *)
	nErrorID							=>,				(* file write error code *)
	sFileName						=>,			(* file name generated from sCaseData *)
	nImigeProcessingSize				=>
);

END_FUNCTION_BLOCK

// ---- POUs/_Exclude/v2_1/FB_CHM_BiuldXMLImige_v2.TcPOU
FUNCTION_BLOCK FB_CHM_BiuldXMLImige_v2
VAR_INPUT
	bExecute					: BOOL;					(* set TRUE to write Case Produced file *)
	hTarget					: UINT;
	eMode						: E_XML_WritingMode;
	nMaxPackItem				: UINT;
	nOuterIndex				: UINT;
	nCodingAndTrackingMode	: UINT;
END_VAR
VAR_IN_OUT
	stAgregationData	 			: ST_CHM_Data;		(* case data to be written to XML *)
END_VAR
VAR_OUTPUT
	bDone						: BOOL;					(* TRUE = XML file write complete *)
	bBusy						: BOOL;					(* TRUE = XML file write in progress *)
	bError						: BOOL;					(* TRUE = XML file write error *)
	nErrorID					: UDINT;				(* file write error code *)
	bVerifyError				: BOOL;					(* TRUE = XML file verification error *)
	nImageByte				: UDINT;
	nWriteImageSize			: UDINT;
END_VAR
VAR
	fbExecute					: R_TRIG;
	eState						: E_XML_CtrlState;
	eErrorState					: E_XML_CtrlState;

	fbWriteFile					: FB_FileWrite;

	bGenerateImage			: BOOL;
	aXMLImage					: ARRAY[0..32767] OF BYTE;
	sString						: T_MaxString;
	nPackIndex				: UINT;
END_VAR

(* rising edge of bExecute triggers new sequence *)
fbExecute(CLK := bExecute);

CASE eState OF

	(* waiting for trigger *)
	E_XML_IDLE:

		(* rising edge of bExecute *)
		IF fbExecute.Q = TRUE THEN

			(* reset internal values *)
			bGenerateImage := FALSE;
			MEMSET(ADR(aXMLImage), 16#00, SIZEOF(aXMLImage));
			nImageByte := 0;
			nWriteImageSize := 0;

			(* update outputs *)
			bBusy := TRUE;
			bDone := FALSE;
			bError := FALSE;
			nErrorID := 0;
			bVerifyError	:= FALSE;

			eErrorState := E_XML_IDLE;

			eState := E_XML_WRITEXML;

		(* bExecute has been reset *)
		ELSIF bExecute = FALSE THEN

			(* update outputs *)
			bBusy := FALSE;
			bDone := FALSE;
			bError := FALSE;
			nErrorID := 0;
			bVerifyError	:= FALSE;
		END_IF

	E_XML_WRITEXML:

		IF NOT bGenerateImage THEN
			CASE eMode OF

				E_CS_HEADER:
					A_CaseHeaderGenerator();

				E_OUTER_HEADER:
					IF nCodingAndTrackingMode >= 7 THEN
						A_OuterHeaderContentGenerator();

						IF nCodingAndTrackingMode = 11 THEN
							FOR nPackIndex := 1 TO nMaxPackItem DO
								A_PackContentGenerator();
							END_FOR
						END_IF

						A_OuterEndPartGenerator();
					END_IF

				E_CS_ENDING:
					A_CaseEndPartGenerator();

			END_CASE

			bGenerateImage := TRUE;
		END_IF

		(* write data to open file *)
		fbWriteFile(
			sNetId		:= '',
			hFile		:= hTarget,
			pWriteBuff	:= ADR(aXMLImage),
			cbWriteLen	:= nImageByte,
			bExecute	:= TRUE,
			tTimeout	:= t#1s
		);

		(* file write completed *)
		IF fbWriteFile.bBusy = FALSE THEN

			(* file write completed OK *)
			IF fbWriteFile.bError = FALSE THEN

				(* log total bytes written *)
				nWriteImageSize := fbWriteFile.cbWrite;

				eState := E_XML_DONE;

			(* file write error *)
			ELSE
				(* no previous error *)
				IF bError = FALSE THEN

					(* log error code and failure state *)
					bError := TRUE;
					nErrorID := fbWriteFile.nErrId;
					eErrorState := eState;
				END_IF

				eState := E_XML_DONE;
			END_IF

			(* close off fbReadFile *)
			fbWriteFile(bExecute := FALSE);
		END_IF

(* sequence complete *)
	E_XML_DONE:

		IF nImageByte <> nWriteImageSize THEN
			bVerifyError := TRUE;
		END_IF

		(* update outputs *)
		bBusy := FALSE;
		bDone := TRUE;

		eState := E_XML_IDLE;
END_CASE

ACTION A_CaseEndPartGenerator:
	IF nCodingAndTrackingMode >= 7 THEN


				(* ItemList end*)
				sString := '$T$T$T$T</ItemList>$R$N';
				MEMMOVE(ADR(aXMLImage[nImageByte]), ADR(sString), LEN(sString));
				nImageByte := nImageByte + LEN(sString);

(***********CASE CONTENT END***********)
			(* Case Content END *)
			sString := '$T$T$T</Content>$R$N';
			MEMMOVE(ADR(aXMLImage[nImageByte]), ADR(sString), LEN(sString));
			nImageByte := nImageByte + LEN(sString);

	END_IF
			(* ProductionOrder *)
			sString := F_CONCAT3('$T$T$T<ProductionOrder>',stAgregationData.GenericHierarchy.CaseItem.ProductionOrder, '</ProductionOrder>$R$N');
			MEMMOVE(ADR(aXMLImage[nImageByte]), ADR(sString), LEN(sString));
			nImageByte := nImageByte + LEN(sString);

			(* LocalProductionOrder *)
			sString := F_CONCAT3('$T$T$T<LocalProductionOrder>',stAgregationData.GenericHierarchy.CaseItem.LocalProductionOrder, '</LocalProductionOrder>$R$N');
			MEMMOVE(ADR(aXMLImage[nImageByte]), ADR(sString), LEN(sString));
			nImageByte := nImageByte + LEN(sString);

			(* PITCode *)
			sString := F_CONCAT3('$T$T$T<PITCode>',stAgregationData.GenericHierarchy.CaseItem.PITCode, '</PITCode>$R$N');
			MEMMOVE(ADR(aXMLImage[nImageByte]), ADR(sString), LEN(sString));
			nImageByte := nImageByte + LEN(sString);

			(* BatchID *)
			sString := F_CONCAT3('$T$T$T<BatchID>',stAgregationData.GenericHierarchy.CaseItem.BatchID, '</BatchID>$R$N');
			MEMMOVE(ADR(aXMLImage[nImageByte]), ADR(sString), LEN(sString));
			nImageByte := nImageByte + LEN(sString);

			(* ProductionLine *)
			sString := F_CONCAT3('$T$T$T<ProductionLine>',stAgregationData.GenericHierarchy.CaseItem.ProductionLine, '</ProductionLine>$R$N');
			MEMMOVE(ADR(aXMLImage[nImageByte]), ADR(sString), LEN(sString));
			nImageByte := nImageByte + LEN(sString);


(***********Item CONTENT END***********)
		(* Item END *)
		sString := '$T$T</Item>$R$N';
		MEMMOVE(ADR(aXMLImage[nImageByte]), ADR(sString), LEN(sString));
		nImageByte := nImageByte + LEN(sString);

(***********GENERIC HIERARCHY CONTENT END***********)

	(* GenericHierarchy END *)
	sString := '$T</GenericHierarchy>$R$N';
	MEMMOVE(ADR(aXMLImage[nImageByte]), ADR(sString), LEN(sString));
	nImageByte := nImageByte + LEN(sString);

	(* Attributes *)
	sString := F_CONCAT3('$T<Attributes>', stAgregationData.Attributes.CSProductionTime, '</Attributes>$R$N');
	MEMMOVE(ADR(aXMLImage[nImageByte]), ADR(sString), LEN(sString));
	nImageByte := nImageByte + LEN(sString);

(* XPath leading tag  END*)
sString := '</GenericHierarchyList> $R$N';
MEMMOVE(ADR(aXMLImage[nImageByte]), ADR(sString), LEN(sString));
nImageByte := nImageByte + LEN(sString);
END_ACTION

ACTION A_CaseHeaderGenerator:
(* XML file version *)
(*sString := '<?xml version="1.0" encoding="utf-8"?>$R$N';
MEMMOVE(ADR(aXMLImage[nImageByte]), ADR(sString), LEN(sString));
nImageByte := nImageByte + LEN(sString);*)

(* XPath leading tag *)
sString := '<GenericHierarchyList xmlns:xsd="http://www.w3.org/2001/XMLSchema" xmlns:xsi="http://www.w3.org/2001/XMLSchema-instance"> $R$N';
MEMMOVE(ADR(aXMLImage[nImageByte]), ADR(sString), LEN(sString));
nImageByte := nImageByte + LEN(sString);

	(* MessageHeader *)
	sString := '$T<MessageHeader>$R$N';
	MEMMOVE(ADR(aXMLImage[nImageByte]), ADR(sString), LEN(sString));
	nImageByte := nImageByte + LEN(sString);

(***********MESSAGE HEADER CONTENT***********)

		(*(* CreationDate *)
		sString := F_CONCAT3('$T$T<CreationDate>',stAgregationData.MessageHeader.CreationDate, '</CreationDate>$R$N');
		MEMMOVE(ADR(aXMLImage[nImageByte]), ADR(sString), LEN(sString));
		nImageByte := nImageByte + LEN(sString);
	
		(* CreationTime *)
		sString := F_CONCAT3('$T$T<CreationTime>',stAgregationData.MessageHeader.CreationTime, '</CreationTime>$R$N');
		MEMMOVE(ADR(aXMLImage[nImageByte]), ADR(sString), LEN(sString));
		nImageByte := nImageByte + LEN(sString);*)

		(* ReferenceID *)
		sString := F_CONCAT3('$T$T<ReferenceID>',stAgregationData.MessageHeader.ReferenceID, '</ReferenceID>$R$N');
		MEMMOVE(ADR(aXMLImage[nImageByte]), ADR(sString), LEN(sString));
		nImageByte := nImageByte + LEN(sString);

		(* CreationTimeLocalUTC *)
		sString := F_CONCAT3('$T$T<CreationTimeLocalUTC>',stAgregationData.MessageHeader.CreationTimeLocalUTC, '</CreationTimeLocalUTC>$R$N');
		MEMMOVE(ADR(aXMLImage[nImageByte]), ADR(sString), LEN(sString));
		nImageByte := nImageByte + LEN(sString);

		(* MessageType *)
		sString := F_CONCAT3('$T$T<MessageType>',stAgregationData.MessageHeader.MessageType, '</MessageType>$R$N');
		MEMMOVE(ADR(aXMLImage[nImageByte]), ADR(sString), LEN(sString));
		nImageByte := nImageByte + LEN(sString);

		(* SenderSystem *)
		sString := F_CONCAT3('$T$T<SenderSystem>',stAgregationData.MessageHeader.SenderSystem, '</SenderSystem>$R$N');
		MEMMOVE(ADR(aXMLImage[nImageByte]), ADR(sString), LEN(sString));
		nImageByte := nImageByte + LEN(sString);

		(* ReceiverSystem *)
		sString := F_CONCAT3('$T$T<ReceiverSystem>',stAgregationData.MessageHeader.ReceiverSystem, '</ReceiverSystem>$R$N');
		MEMMOVE(ADR(aXMLImage[nImageByte]), ADR(sString), LEN(sString));
		nImageByte := nImageByte + LEN(sString);

(***********MESSAGE HEADER CONTENT END***********)

	(* MessageHeader END *)
	sString := '$T</MessageHeader>$R$N';
	MEMMOVE(ADR(aXMLImage[nImageByte]), ADR(sString), LEN(sString));
	nImageByte := nImageByte + LEN(sString);

	(* Factory*)
	sString := F_CONCAT3('$T<Factory>', stAgregationData.Factory, '</Factory>$R$N');
	MEMMOVE(ADR(aXMLImage[nImageByte]), ADR(sString), LEN(sString));
	nImageByte := nImageByte + LEN(sString);

	(* GenericHierarchy *)
	sString := '$T<GenericHierarchy>$R$N';
	MEMMOVE(ADR(aXMLImage[nImageByte]), ADR(sString), LEN(sString));
	nImageByte := nImageByte + LEN(sString);

(***********GENERIC HIERARCHY CONTENT***********)

		(* HierarchyType *)
		sString := F_CONCAT3('$T$T<HierarchyType>',stAgregationData.GenericHierarchy.HierarchyType, '</HierarchyType>$R$N');
		MEMMOVE(ADR(aXMLImage[nImageByte]), ADR(sString), LEN(sString));
		nImageByte := nImageByte + LEN(sString);

		(* PerformedAction *)
		sString := F_CONCAT3('$T$T<ACTION>',stAgregationData.GenericHierarchy.PerformedAction, '</ACTION>$R$N');
		MEMMOVE(ADR(aXMLImage[nImageByte]), ADR(sString), LEN(sString));
		nImageByte := nImageByte + LEN(sString);

		(* TrackingLevels *)
		sString := F_CONCAT3('$T$T<TrackingLevels>',stAgregationData.GenericHierarchy.TrackingLevels, '</TrackingLevels>$R$N');
		MEMMOVE(ADR(aXMLImage[nImageByte]), ADR(sString), LEN(sString));
		nImageByte := nImageByte + LEN(sString);

		(* TrackingIndicator *)
		sString := F_CONCAT3('$T$T<TrackingIndicator>',stAgregationData.GenericHierarchy.TrackingIndicator, '</TrackingIndicator>$R$N');
		MEMMOVE(ADR(aXMLImage[nImageByte]), ADR(sString), LEN(sString));
		nImageByte := nImageByte + LEN(sString);

		(* Item Type *)
		sString := '$T$T<Item Type="CS">$R$N';
		MEMMOVE(ADR(aXMLImage[nImageByte]), ADR(sString), LEN(sString));
		nImageByte := nImageByte + LEN(sString);

(***********Item Type CONTENT***********)
			(* Identity*)
			sString := '$T$T$T<Identity>$R$N';
			MEMMOVE(ADR(aXMLImage[nImageByte]), ADR(sString), LEN(sString));
			nImageByte := nImageByte + LEN(sString);

(***********Identity CONTENT***********)
					(* SKU *)
					sString := F_CONCAT3('$T$T$T$T<SKU>',stAgregationData.GenericHierarchy.CaseItem.Identity.SKU, '</SKU>$R$N');
					MEMMOVE(ADR(aXMLImage[nImageByte]), ADR(sString), LEN(sString));
					nImageByte := nImageByte + LEN(sString);

					(* GTIN *)
					sString := F_CONCAT3('$T$T$T$T<GTIN>',stAgregationData.GenericHierarchy.CaseItem.Identity.GTIN, '</GTIN>$R$N');
					MEMMOVE(ADR(aXMLImage[nImageByte]), ADR(sString), LEN(sString));
					nImageByte := nImageByte + LEN(sString);

					(* ID *)
					sString := F_CONCAT3('$T$T$T$T<ID>',stAgregationData.GenericHierarchy.CaseItem.Identity.ID, '</ID>$R$N');
					MEMMOVE(ADR(aXMLImage[nImageByte]), ADR(sString), LEN(sString));
					nImageByte := nImageByte + LEN(sString);

					(* ReadQuality *)
					sString := F_CONCAT3('$T$T$T$T<ReadQuality>',stAgregationData.GenericHierarchy.CaseItem.Identity.ReadQuality, '</ReadQuality>$R$N');
					MEMMOVE(ADR(aXMLImage[nImageByte]), ADR(sString), LEN(sString));
					nImageByte := nImageByte + LEN(sString);

(***********Identity CONTENT END***********)

			(* Identity END *)
			sString := '$T$T$T</Identity>$R$N';
			MEMMOVE(ADR(aXMLImage[nImageByte]), ADR(sString), LEN(sString));
			nImageByte := nImageByte + LEN(sString);

			(* ItemState *)
			sString := F_CONCAT3('$T$T$T<ItemState>',stAgregationData.GenericHierarchy.CaseItem.ItemState, '</ItemState>$R$N');
			MEMMOVE(ADR(aXMLImage[nImageByte]), ADR(sString), LEN(sString));
			nImageByte := nImageByte + LEN(sString);

			(* RejectReason *)
			sString := '$T$T$T<RejectReason>$R$N';
			MEMMOVE(ADR(aXMLImage[nImageByte]), ADR(sString), LEN(sString));
			nImageByte := nImageByte + LEN(sString);

				sString := F_CONCAT3('$T$T$T$T<Reason>',stAgregationData.GenericHierarchy.CaseItem.RejectReason, '</Reason>$R$N');
				MEMMOVE(ADR(aXMLImage[nImageByte]), ADR(sString), LEN(sString));
				nImageByte := nImageByte + LEN(sString);

			sString := '$T$T$T</RejectReason>$R$N';
			MEMMOVE(ADR(aXMLImage[nImageByte]), ADR(sString), LEN(sString));
			nImageByte := nImageByte + LEN(sString);

			(*logs *)
			sString := '$T$T$T<logs>$R$N';
			MEMMOVE(ADR(aXMLImage[nImageByte]), ADR(sString), LEN(sString));
			nImageByte := nImageByte + LEN(sString);

				(* TimeStamp *)
				sString := F_CONCAT3('$T$T$T$T<TimeStamp Topic="Aggregation">',stAgregationData.GenericHierarchy.CaseItem.TimeStamp, '</TimeStamp>$R$N');
				MEMMOVE(ADR(aXMLImage[nImageByte]), ADR(sString), LEN(sString));
				nImageByte := nImageByte + LEN(sString);

			(* logs END *)
			sString := '$T$T$T</logs>$R$N';
			MEMMOVE(ADR(aXMLImage[nImageByte]), ADR(sString), LEN(sString));
			nImageByte := nImageByte + LEN(sString);

			(* NoRead *)
			sString := F_CONCAT3('$T$T$T<NoRead>',stAgregationData.GenericHierarchy.CaseItem.NoRead, '</NoRead>$R$N');
			MEMMOVE(ADR(aXMLImage[nImageByte]), ADR(sString), LEN(sString));
			nImageByte := nImageByte + LEN(sString);

(***********CONTENT***********)
	IF nCodingAndTrackingMode >= 7 THEN

			(* Case Content *)
			sString := '$T$T$T<Content>$R$N';
			MEMMOVE(ADR(aXMLImage[nImageByte]), ADR(sString), LEN(sString));
			nImageByte := nImageByte + LEN(sString);

				(* Case DefaultIdentity*)
				sString := '$T$T$T$T<DefaultIdentity>$R$N';
				MEMMOVE(ADR(aXMLImage[nImageByte]), ADR(sString), LEN(sString));
				nImageByte := nImageByte + LEN(sString);

						(* SKU *)
						sString := F_CONCAT3('$T$T$T$T$T<SKU>',stAgregationData.GenericHierarchy.CaseItem.Content.DefaultIdentity.SKU, '</SKU>$R$N');
						MEMMOVE(ADR(aXMLImage[nImageByte]), ADR(sString), LEN(sString));
						nImageByte := nImageByte + LEN(sString);

						(* GTIN *)
						sString := F_CONCAT3('$T$T$T$T$T<GTIN>',stAgregationData.GenericHierarchy.CaseItem.Content.DefaultIdentity.GTIN, '</GTIN>$R$N');
						MEMMOVE(ADR(aXMLImage[nImageByte]), ADR(sString), LEN(sString));
						nImageByte := nImageByte + LEN(sString);

						(* ProductionOrder *)
						sString := F_CONCAT3('$T$T$T$T$T<ProductionOrder>',stAgregationData.GenericHierarchy.CaseItem.Content.DefaultIdentity.ProductionOrder, '</ProductionOrder>$R$N');
						MEMMOVE(ADR(aXMLImage[nImageByte]), ADR(sString), LEN(sString));
						nImageByte := nImageByte + LEN(sString);

						(* LocalProductionOrder *)
						sString := F_CONCAT3('$T$T$T$T$T<LocalProductionOrder>',stAgregationData.GenericHierarchy.CaseItem.Content.DefaultIdentity.LocalProductionOrder, '</LocalProductionOrder>$R$N');
						MEMMOVE(ADR(aXMLImage[nImageByte]), ADR(sString), LEN(sString));
						nImageByte := nImageByte + LEN(sString);

						(* PITCode *)
						sString := F_CONCAT3('$T$T$T$T$T<PITCode>',stAgregationData.GenericHierarchy.CaseItem.Content.DefaultIdentity.PITCode, '</PITCode>$R$N');
						MEMMOVE(ADR(aXMLImage[nImageByte]), ADR(sString), LEN(sString));
						nImageByte := nImageByte + LEN(sString);

						(* BatchID *)
						sString := F_CONCAT3('$T$T$T$T$T<BatchID>',stAgregationData.GenericHierarchy.CaseItem.Content.DefaultIdentity.BatchID, '</BatchID>$R$N');
						MEMMOVE(ADR(aXMLImage[nImageByte]), ADR(sString), LEN(sString));
						nImageByte := nImageByte + LEN(sString);

						(* ProductionLine *)
						sString := F_CONCAT3('$T$T$T$T$T<ProductionLine>',stAgregationData.GenericHierarchy.CaseItem.Content.DefaultIdentity.ProductionLine, '</ProductionLine>$R$N');
						MEMMOVE(ADR(aXMLImage[nImageByte]), ADR(sString), LEN(sString));
						nImageByte := nImageByte + LEN(sString);

				(* Case DefaultIdentity END*)
				sString := '$T$T$T$T</DefaultIdentity>$R$N';
				MEMMOVE(ADR(aXMLImage[nImageByte]), ADR(sString), LEN(sString));
				nImageByte := nImageByte + LEN(sString);

				(* ExpectedItemCount *)
				sString := F_CONCAT3('$T$T$T$T<ExpectedItemCount>',stAgregationData.GenericHierarchy.CaseItem.Content.ExpectedItemCount, '</ExpectedItemCount>$R$N');
				MEMMOVE(ADR(aXMLImage[nImageByte]), ADR(sString), LEN(sString));
				nImageByte := nImageByte + LEN(sString);

				(* ItemReadRate *)
				sString := F_CONCAT3('$T$T$T$T<ItemReadRate>',stAgregationData.GenericHierarchy.CaseItem.Content.ItemReadRate, '</ItemReadRate>$R$N');
				MEMMOVE(ADR(aXMLImage[nImageByte]), ADR(sString), LEN(sString));
				nImageByte := nImageByte + LEN(sString);

				(* ItemList*)
				sString := '$T$T$T$T<ItemList>$R$N';
				MEMMOVE(ADR(aXMLImage[nImageByte]), ADR(sString), LEN(sString));
				nImageByte := nImageByte + LEN(sString);
	END_IF
END_ACTION

ACTION A_OuterEndPartGenerator:
(*
    </ItemList> 
                        </Content> 
                    </Item> 

*)
						IF nCodingAndTrackingMode = 11 THEN
								(* ItemList end*)
								sString := '$T$T$T$T$T$T$T</ItemList>$R$N';
								MEMMOVE(ADR(aXMLImage[nImageByte]), ADR(sString), LEN(sString));
								nImageByte := nImageByte + LEN(sString);
	(***********CASE CONTENT END***********)
							(* Outer Content END *)
							sString := '$T$T$T$T$T$T</Content>$R$N';
							MEMMOVE(ADR(aXMLImage[nImageByte]), ADR(sString), LEN(sString));
							nImageByte := nImageByte + LEN(sString);
						END_IF

								(* Item Type END *)
								sString := '$T$T$T$T$T</Item>$R$N';
							MEMMOVE(ADR(aXMLImage[nImageByte]), ADR(sString), LEN(sString));
							nImageByte := nImageByte + LEN(sString);
END_ACTION

ACTION A_OuterHeaderContentGenerator:
(*
                  <Item Type="OUT"> 
                        <Identity> 
                         	   <ID>55128CY203644964300</ID> 
                        	    <ReadQuality>100</ReadQuality> 
                        </Identity> 
                        <ItemState>Verified</ItemState> 
                        <RejectReason /> 
                        <logs> 
                   		        <TimeStamp Topic="Aggregation">2018-03-22T20:46:01.5229666+01:00</TimeStamp> 
                        </logs> 
                        <NoRead>false</NoRead> 
                        <Content> 
                           	 <DefaultIdentity> 
                      	     	     <SKU>10045622</SKU> 
                        	   	     <GTIN>00000087295993</GTIN> 
                        		        <ProductionOrder>2523549</ProductionOrder> 
                         		       <LocalProductionOrder>2523549</LocalProductionOrder> 
                           		     <PITCode>3</PITCode> 
                          		      <BatchID>55122018</BatchID> 
                        		        <ProductionLine>12</ProductionLine> 
                       	     </DefaultIdentity> 
                      	      <ExpectedItemCount>10</ExpectedItemCount> 
                       	     <ItemReadRate>100</ItemReadRate> 
                       	     <ItemList> 

*)


					(* Item Type *)
					sString := '$T$T$T$T$T<Item Type="OUT">$R$N';
					MEMMOVE(ADR(aXMLImage[nImageByte]), ADR(sString), LEN(sString));
					nImageByte := nImageByte + LEN(sString);

						(* Identity *)
						sString := '$T$T$T$T$T$T<Identity>$R$N';
						MEMMOVE(ADR(aXMLImage[nImageByte]), ADR(sString), LEN(sString));
						nImageByte := nImageByte + LEN(sString);

							(* ID *)
							sString := F_CONCAT3('$T$T$T$T$T$T$T<ID><![CDATA[',stAgregationData.GenericHierarchy.CaseItem.Content.arrOuterItem[nOuterIndex].Identity.ID, ']]></ID>$R$N');
							MEMMOVE(ADR(aXMLImage[nImageByte]), ADR(sString), LEN(sString));
							nImageByte := nImageByte + LEN(sString);

							(* ReadQuality *)
							sString := F_CONCAT3('$T$T$T$T$T$T$T<ReadQuality>',stAgregationData.GenericHierarchy.CaseItem.Content.arrOuterItem[nOuterIndex].Identity.ReadQuality, '</ReadQuality>$R$N');
							MEMMOVE(ADR(aXMLImage[nImageByte]), ADR(sString), LEN(sString));
							nImageByte := nImageByte + LEN(sString);

						(* Identity END *)
						sString := '$T$T$T$T$T$T</Identity>$R$N';
						MEMMOVE(ADR(aXMLImage[nImageByte]), ADR(sString), LEN(sString));
						nImageByte := nImageByte + LEN(sString);


						(* ItemState *)
						sString := F_CONCAT3('$T$T$T$T$T$T<ItemState>',stAgregationData.GenericHierarchy.CaseItem.Content.arrOuterItem[nOuterIndex].ItemState, '</ItemState>$R$N');
						MEMMOVE(ADR(aXMLImage[nImageByte]), ADR(sString), LEN(sString));
						nImageByte := nImageByte + LEN(sString);

						(* RejectReason *)
						sString := '$T$T$T$T$T$T<RejectReason>$R$N';
						MEMMOVE(ADR(aXMLImage[nImageByte]), ADR(sString), LEN(sString));
						nImageByte := nImageByte + LEN(sString);
			
							sString := F_CONCAT3('$T$T$T$T$T$T$T<Reason>',stAgregationData.GenericHierarchy.CaseItem.Content.arrOuterItem[nOuterIndex].RejectReason, '</Reason>$R$N');
							MEMMOVE(ADR(aXMLImage[nImageByte]), ADR(sString), LEN(sString));
							nImageByte := nImageByte + LEN(sString);
			
						sString := '$T$T$T$T$T$T</RejectReason>$R$N';
						MEMMOVE(ADR(aXMLImage[nImageByte]), ADR(sString), LEN(sString));
						nImageByte := nImageByte + LEN(sString);


						(*logs *)
						sString := '$T$T$T$T$T$T<logs>$R$N';
						MEMMOVE(ADR(aXMLImage[nImageByte]), ADR(sString), LEN(sString));
						nImageByte := nImageByte + LEN(sString);

							(* TimeStamp *)
							sString := F_CONCAT3('$T$T$T$T$T$T$T<TimeStamp Topic="Aggregation">',stAgregationData.GenericHierarchy.CaseItem.Content.arrOuterItem[nOuterIndex].TimeStamp, '</TimeStamp>$R$N');
							MEMMOVE(ADR(aXMLImage[nImageByte]), ADR(sString), LEN(sString));
							nImageByte := nImageByte + LEN(sString);

						(* logs END *)
						sString := '$T$T$T$T$T$T</logs>$R$N';
						MEMMOVE(ADR(aXMLImage[nImageByte]), ADR(sString), LEN(sString));
						nImageByte := nImageByte + LEN(sString);

						(* NoRead *)
						sString := F_CONCAT3('$T$T$T$T$T$T<NoRead>',stAgregationData.GenericHierarchy.CaseItem.Content.arrOuterItem[nOuterIndex].NoRead, '</NoRead>$R$N');
						MEMMOVE(ADR(aXMLImage[nImageByte]), ADR(sString), LEN(sString));
						nImageByte := nImageByte + LEN(sString);
(***********CONTENT***********)

						IF nCodingAndTrackingMode = 11 THEN
							(* Outer Content *)
							sString := '$T$T$T$T$T$T<Content>$R$N';
							MEMMOVE(ADR(aXMLImage[nImageByte]), ADR(sString), LEN(sString));
							nImageByte := nImageByte + LEN(sString);
	
	
								(* Case DefaultIdentity*)
								sString := '$T$T$T$T$T$T$T<DefaultIdentity>$R$N';
								MEMMOVE(ADR(aXMLImage[nImageByte]), ADR(sString), LEN(sString));
								nImageByte := nImageByte + LEN(sString);
	
										(* SKU *)
										sString := F_CONCAT3('$T$T$T$T$T$T$T$T<SKU>',stAgregationData.GenericHierarchy.CaseItem.Content.arrOuterItem[nOuterIndex].Content.DefaultIdentity.SKU, '</SKU>$R$N');
										MEMMOVE(ADR(aXMLImage[nImageByte]), ADR(sString), LEN(sString));
										nImageByte := nImageByte + LEN(sString);
	
										(* GTIN *)
										sString := F_CONCAT3('$T$T$T$T$T$T$T$T<GTIN>',stAgregationData.GenericHierarchy.CaseItem.Content.arrOuterItem[nOuterIndex].Content.DefaultIdentity.GTIN, '</GTIN>$R$N');
										MEMMOVE(ADR(aXMLImage[nImageByte]), ADR(sString), LEN(sString));
										nImageByte := nImageByte + LEN(sString);
	
										(* ProductionOrder *)
										sString := F_CONCAT3('$T$T$T$T$T$T$T$T<ProductionOrder>',stAgregationData.GenericHierarchy.CaseItem.Content.arrOuterItem[nOuterIndex].Content.DefaultIdentity.ProductionOrder, '</ProductionOrder>$R$N');
										MEMMOVE(ADR(aXMLImage[nImageByte]), ADR(sString), LEN(sString));
										nImageByte := nImageByte + LEN(sString);
	
										(* LocalProductionOrder *)
										sString := F_CONCAT3('$T$T$T$T$T$T$T$T<LocalProductionOrder>',stAgregationData.GenericHierarchy.CaseItem.Content.arrOuterItem[nOuterIndex].Content.DefaultIdentity.LocalProductionOrder, '</LocalProductionOrder>$R$N');
										MEMMOVE(ADR(aXMLImage[nImageByte]), ADR(sString), LEN(sString));
										nImageByte := nImageByte + LEN(sString);
	
										(* PITCode *)
										sString := F_CONCAT3('$T$T$T$T$T$T$T$T<PITCode>',stAgregationData.GenericHierarchy.CaseItem.Content.arrOuterItem[nOuterIndex].Content.DefaultIdentity.PITCode, '</PITCode>$R$N');
										MEMMOVE(ADR(aXMLImage[nImageByte]), ADR(sString), LEN(sString));
										nImageByte := nImageByte + LEN(sString);
	
										(* BatchID *)
										sString := F_CONCAT3('$T$T$T$T$T$T$T$T<BatchID>',stAgregationData.GenericHierarchy.CaseItem.Content.arrOuterItem[nOuterIndex].Content.DefaultIdentity.BatchID, '</BatchID>$R$N');
										MEMMOVE(ADR(aXMLImage[nImageByte]), ADR(sString), LEN(sString));
										nImageByte := nImageByte + LEN(sString);
	
										(* ProductionLine *)
										sString := F_CONCAT3('$T$T$T$T$T$T$T$T<ProductionLine>',stAgregationData.GenericHierarchy.CaseItem.Content.arrOuterItem[nOuterIndex].Content.DefaultIdentity.ProductionLine, '</ProductionLine>$R$N');
										MEMMOVE(ADR(aXMLImage[nImageByte]), ADR(sString), LEN(sString));
										nImageByte := nImageByte + LEN(sString);
	
								(* Case DefaultIdentity END*)
								sString := '$T$T$T$T$T$T$T</DefaultIdentity>$R$N';
								MEMMOVE(ADR(aXMLImage[nImageByte]), ADR(sString), LEN(sString));
								nImageByte := nImageByte + LEN(sString);
	
								(* ExpectedItemCount *)
								sString := F_CONCAT3('$T$T$T$T$T$T$T<ExpectedItemCount>',stAgregationData.GenericHierarchy.CaseItem.Content.arrOuterItem[nOuterIndex].Content.ExpectedItemCount, '</ExpectedItemCount>$R$N');
								MEMMOVE(ADR(aXMLImage[nImageByte]), ADR(sString), LEN(sString));
								nImageByte := nImageByte + LEN(sString);
	
								(* ItemReadRate *)
								sString := F_CONCAT3('$T$T$T$T$T$T$T<ItemReadRate>',stAgregationData.GenericHierarchy.CaseItem.Content.arrOuterItem[nOuterIndex].Content.ItemReadRate, '</ItemReadRate>$R$N');
								MEMMOVE(ADR(aXMLImage[nImageByte]), ADR(sString), LEN(sString));
								nImageByte := nImageByte + LEN(sString);
	
								(* ItemList*)
								sString := '$T$T$T$T$T$T$T<ItemList>$R$N';
								MEMMOVE(ADR(aXMLImage[nImageByte]), ADR(sString), LEN(sString));
								nImageByte := nImageByte + LEN(sString);
						END_IF
END_ACTION

ACTION A_PackContentGenerator:
(*
                             <Item Type="PK"> 
                                    <Identity> 
                                        <ID>1XJWVXUS1FM7</ID> 
                                        <ReadQuality>100</ReadQuality> 
                                    </Identity> 
                                    <ItemState>Verified</ItemState> 
                                    <RejectReason /> 
                                    <logs> 
                                        <TimeStamp Topic="Aggregation">2018-03-22T20:45:38.4129952+01:00</TimeStamp> 
                                    </logs> 
                                    <NoRead>false</NoRead> 
                                </Item> 
*)

								(* Item Type *)
								sString := '$T$T$T$T$T$T$T$T<Item Type="PK">$R$N';
								MEMMOVE(ADR(aXMLImage[nImageByte]), ADR(sString), LEN(sString));
								nImageByte := nImageByte + LEN(sString);

									(* Identity *)
									sString := '$T$T$T$T$T$T$T$T$T<Identity>$R$N';
									MEMMOVE(ADR(aXMLImage[nImageByte]), ADR(sString), LEN(sString));
									nImageByte := nImageByte + LEN(sString);

										(* ID *)
										sString := F_CONCAT3('$T$T$T$T$T$T$T$T$T$T<ID><![CDATA[',stAgregationData.GenericHierarchy.CaseItem.Content.arrOuterItem[nOuterIndex].Content.arrPackItem[nPackIndex].Identity.ID, ']]></ID>$R$N');
										MEMMOVE(ADR(aXMLImage[nImageByte]), ADR(sString), LEN(sString));
										nImageByte := nImageByte + LEN(sString);

										(* ReadQuality *)
										sString := F_CONCAT3('$T$T$T$T$T$T$T$T$T$T<ReadQuality>',stAgregationData.GenericHierarchy.CaseItem.Content.arrOuterItem[nOuterIndex].Content.arrPackItem[nPackIndex].Identity.ReadQuality, '</ReadQuality>$R$N');
										MEMMOVE(ADR(aXMLImage[nImageByte]), ADR(sString), LEN(sString));
										nImageByte := nImageByte + LEN(sString);

									(* Identity END *)
									sString := '$T$T$T$T$T$T$T$T$T</Identity>$R$N';
									MEMMOVE(ADR(aXMLImage[nImageByte]), ADR(sString), LEN(sString));
									nImageByte := nImageByte + LEN(sString);

									(* ItemState *)
									sString := F_CONCAT3('$T$T$T$T$T$T$T$T$T<ItemState>',stAgregationData.GenericHierarchy.CaseItem.Content.arrOuterItem[nOuterIndex].Content.arrPackItem[nPackIndex].ItemState, '</ItemState>$R$N');
									MEMMOVE(ADR(aXMLImage[nImageByte]), ADR(sString), LEN(sString));
									nImageByte := nImageByte + LEN(sString);
			

									(* RejectReason *)
									sString := '$T$T$T$T$T$T$T$T$T<RejectReason>$R$N';
									MEMMOVE(ADR(aXMLImage[nImageByte]), ADR(sString), LEN(sString));
									nImageByte := nImageByte + LEN(sString);

										sString := F_CONCAT3('$T$T$T$T$T$T$T$T$T$T<Reason>',stAgregationData.GenericHierarchy.CaseItem.Content.arrOuterItem[nOuterIndex].Content.arrPackItem[nPackIndex].RejectReason, '</Reason>$R$N');
										MEMMOVE(ADR(aXMLImage[nImageByte]), ADR(sString), LEN(sString));
										nImageByte := nImageByte + LEN(sString);
			
									sString := '$T$T$T$T$T$T$T$T$T</RejectReason>$R$N';
									MEMMOVE(ADR(aXMLImage[nImageByte]), ADR(sString), LEN(sString));
									nImageByte := nImageByte + LEN(sString);


									(*logs *)
									sString := '$T$T$T$T$T$T$T$T$T<logs>$R$N';
									MEMMOVE(ADR(aXMLImage[nImageByte]), ADR(sString), LEN(sString));
									nImageByte := nImageByte + LEN(sString);
	
										(* TimeStamp *)
										sString := F_CONCAT3('$T$T$T$T$T$T$T$T$T$T<TimeStamp Topic="Aggregation">',stAgregationData.GenericHierarchy.CaseItem.Content.arrOuterItem[nOuterIndex].Content.arrPackItem[nPackIndex].TimeStamp, '</TimeStamp>$R$N');
										MEMMOVE(ADR(aXMLImage[nImageByte]), ADR(sString), LEN(sString));
										nImageByte := nImageByte + LEN(sString);
			
									(* logs END *)
									sString := '$T$T$T$T$T$T$T$T$T</logs>$R$N';
									MEMMOVE(ADR(aXMLImage[nImageByte]), ADR(sString), LEN(sString));
									nImageByte := nImageByte + LEN(sString);

									(* No Read *)
									sString := F_CONCAT3('$T$T$T$T$T$T$T$T$T<NoRead>',stAgregationData.GenericHierarchy.CaseItem.Content.arrOuterItem[nOuterIndex].Content.arrPackItem[nPackIndex].NoRead, '</NoRead>$R$N');
									MEMMOVE(ADR(aXMLImage[nImageByte]), ADR(sString), LEN(sString));
									nImageByte := nImageByte + LEN(sString);

								(* Item Type END *)
								sString := '$T$T$T$T$T$T$T$T</Item>$R$N';
								MEMMOVE(ADR(aXMLImage[nImageByte]), ADR(sString), LEN(sString));
								nImageByte := nImageByte + LEN(sString);
END_ACTION

END_FUNCTION_BLOCK

// ---- POUs/_Exclude/v2_1/FB_CHM_HierachyGenerator.TcPOU
FUNCTION_BLOCK FB_CHM_HierachyGenerator
VAR_INPUT
	bExecute						: BOOL;
	sLocalCHMPath				: STRING(50);
	sCHMFileName					: T_CHM_Filename;	(* current PCM file *)
	nMaxOuterItem				: UINT	:=cMAX_OUTERS_PER_CASE;
	nMaxPackItem					: UINT	:=cMAX_PACKS_PER_OUTER;
	bClearStatistic					: BOOL;
	nCodingAndTrackingMode		: UINT;
	tTimeOut						: TIME;
	bIsValid						: BOOL;
END_VAR
VAR_IN_OUT
	stCHMDataStruct				: ST_CHM_Data;
END_VAR
VAR_OUTPUT
	bDone							: BOOL;					(* TRUE = XML file write complete *)
	bBusy							: BOOL;					(* TRUE = XML file write in progress *)
	bError							: BOOL;					(* TRUE = XML file write error *)
	nErrorID						: UDINT;				(* file write error code *)
	stLastCaseHierarchyMessage	: ST_CHM_Data;
	nLastImigeSize					: UDINT;
	tPerformanceRate				 :TIME;
END_VAR
VAR
	eStep					: E_CHM_GeneratorState;
	eErrorState				: E_CHM_GeneratorState;

	rtrigExecute			: R_TRIG;
	rtrigFBDone			: R_TRIG;

	tonTimeOut			: TON;
	tonPerfomance			: TON;

	(*pWriteBuffer		: UDINT;
	nWriteBytes			: UDINT;*)

	eCommand				: E_EnumCmdType;
	fbFindFile				: FB_EnumFindFileEntry;
	strFoundFile			: T_MaxString;

	hTarget				: UINT;
	fbOpenFile				: FB_FileOpen;
	fbCloseFile				: FB_FileClose;

	eCurrentXMLMode			:  E_XML_WritingMode;
	fbWriteCHMDataToXML	: FB_CHM_BiuldXMLImige_v2;

	bSkipFLGFile				: BOOL;
	fbCreateFLGFile			: FB_CHM_SaveFLG_File;

	aImigeSize			:	 ARRAY[0..100] OF UDINT;

	nCHMOuterIndex		: 	UINT := 1;
	nMaxCHMOuterIndex	: 	UINT;

	bWriteCaseDataToXML	:	BOOL;
	bCreatFLGFileExe		: 	BOOL;

	nSequenceNumber		: 	INT;

END_VAR

rtrigExecute(CLK:=bExecute);

tonTimeOut(IN:= bBusy, PT:= tTimeOut);

IF tonTimeOut.Q AND tTimeOut <> t#0ms THEN

	bDone	:=  	TRUE;
	bBusy	:=  	FALSE;
	bError	:= 	TRUE;
	nErrorID	:= 	1;

	hTarget				:= 0;
	bSkipFLGFile			:= FALSE;

	bWriteCaseDataToXML	:= FALSE;
	bCreatFLGFileExe		:= FALSE;

	tPerformanceRate 	:= tonPerfomance.ET;
	eErrorState			:= E_CHM_TIMEOUT;

	eStep	:= E_CHM_IDLEGENERATOR;
END_IF

tonPerfomance(IN:= eStep<>E_CHM_IDLEGENERATOR, PT:= t#30s);

IF bClearStatistic THEN
	MEMSET(ADR(aImigeSize), 16#00, SIZEOF(aImigeSize));
END_IF

CASE eStep OF

	E_CHM_IDLEGENERATOR:
	
		IF rtrigExecute.Q THEN

			(* update outputs *)
			bDone := FALSE;
			bBusy := TRUE;
			bError := FALSE;
			nErrorID := 0;

			eCommand 	:= eEnumCmd_First;
			strFoundFile	:= '';

			nCHMOuterIndex		:= 1;
			hTarget				:= 0;
			bWriteCaseDataToXML	:= FALSE;
			bCreatFLGFileExe		:= FALSE;
			bSkipFLGFile			:= FALSE;

			MEMSET(ADR(stLastCaseHierarchyMessage), 16#00, SIZEOF(stLastCaseHierarchyMessage));
	
			nLastImigeSize		:= 0;
			tPerformanceRate	 :=t#0ms;
			eErrorState			:= E_CHM_IDLEGENERATOR;

			eStep	:=E_CHM_FILECHECK;

		ELSIF NOT bExecute THEN

			bDone 	:= FALSE;
			bBusy 	:= FALSE;
			bError 	:= FALSE;
			nErrorID	 := 0;
	
			hTarget		:= 0;
			bSkipFLGFile	:= FALSE;
			
			bWriteCaseDataToXML	:= FALSE;
			bCreatFLGFileExe		:= FALSE;

			strFoundFile	:= '';

		END_IF

(* find file *)
	E_CHM_FILECHECK:

		(* get file name *)
		fbFindFile(
			sNetId		:= '',
			sPathName	:= CONCAT(sLocalCHMPath, sCHMFileName),
			eCmd		:= eCommand,
			bExecute	:= TRUE,
			tTimeout	:= T#1s,
		);

		(* find file complete *)
		IF fbFindFile.bBusy = FALSE THEN

			(* find file completed OK *)
			IF fbFindFile.bError = FALSE THEN

				(* file found *)
				IF fbFindFile.bEOE = FALSE THEN

					(* ignore filenames '.' and '..' *)
					IF fbFindFile.stFindFile.sFileName <> '.' AND fbFindFile.stFindFile.sFileName <> '..' THEN
						strFoundFile := fbFindFile.stFindFile.sFileName;
					END_IF
					eStep := E_CHM_DONEGENERATOR;
				(* end of file list *)
				ELSE
					(* copy files complete *)
					eStep := E_CHM_FILEOPEN;
				END_IF
			(* find file error *)
			ELSE

				(* no error has previously occurred *)
				IF bError = FALSE THEN

					(* log error code and failure state *)
					bError := TRUE;
					nErrorID := fbFindFile.nErrId;
					eErrorState := eStep;
				END_IF

				(* abandon attempt to copy files *)
				eStep := E_CHM_DONEGENERATOR;
			END_IF

			(* close off fbFindFile *)
			fbFindFile(bExecute := FALSE);
		END_IF

	E_CHM_FILEOPEN:
	(* open file for writing in binary mode *)
		fbOpenFile(
			sNetId		:= '',
			sPathName	:=  CONCAT(sLocalCHMPath, sCHMFileName),
			nMode		:= FOPEN_MODEAPPEND OR FOPEN_MODEPLUS OR FOPEN_MODEBINARY,
			ePath		:= PATH_GENERIC,
			bExecute	:= TRUE,
			tTimeout	:= T#1s
		);

		(* file open completed *)
		IF fbOpenFile.bBusy = FALSE THEN

			(* file open completed OK *)
			IF fbOpenFile.bError = FALSE THEN

				(* log file handle for use by subsequent commands *)
				hTarget := fbOpenFile.hFile;

				eStep := E_CHM_GENERATEHEAD;

			(* file open error *)
			ELSE

				(* log error code and failure state *)
				bError := TRUE;
				nErrorID := fbOpenFile.nErrId;
				eErrorState := eStep;

				(* abandon attempt to read file *)
				eStep := E_CHM_DONEGENERATOR;
			END_IF

			(* close off fbOpenFile *)
			fbOpenFile(bExecute := FALSE);
		END_IF

	E_CHM_GENERATEHEAD:

		MEMSET(ADR(aImigeSize), 16#00, SIZEOF(aImigeSize));

		bWriteCaseDataToXML := TRUE;
		eCurrentXMLMode := E_CS_HEADER;

		IF fbWriteCHMDataToXML.bDone THEN

			IF NOT fbWriteCHMDataToXML.bError THEN

				eStep	:=E_CHM_GENERATEBODY;
			ELSE

				bError 	:= TRUE;
				nErrorID	 := fbWriteCHMDataToXML.nErrorID;
				bSkipFLGFile			:= TRUE;

				eErrorState := eStep;

				eStep	:=E_CHM_FILECLOSE;
			END_IF

			bWriteCaseDataToXML := FALSE;
		END_IF

	E_CHM_GENERATEBODY:

		bWriteCaseDataToXML := TRUE;
		eCurrentXMLMode := E_OUTER_HEADER;

		IF fbWriteCHMDataToXML.bDone THEN

			IF NOT fbWriteCHMDataToXML.bError THEN

				IF nCHMOuterIndex >= nMaxOuterItem  THEN
			
					eStep	:=E_CHM_GENERATEENDING;
				ELSE
					nCHMOuterIndex	:=	nCHMOuterIndex+1;
					eStep	:=E_CHM_GENERATEBODY;
				END_IF

			ELSE

				bError 	:= TRUE;
				nErrorID	 := fbWriteCHMDataToXML.nErrorID;
				bSkipFLGFile			:= TRUE;
	
				eErrorState := eStep;
		
				eStep	:=E_CHM_FILECLOSE;
			END_IF

			bWriteCaseDataToXML := FALSE;
		END_IF

	E_CHM_GENERATEENDING:
	
		bWriteCaseDataToXML := TRUE;
		eCurrentXMLMode := E_CS_ENDING;

		IF fbWriteCHMDataToXML.bDone THEN

			IF NOT	fbWriteCHMDataToXML.bError	THEN
				nMaxCHMOuterIndex	:= nCHMOuterIndex;
				nCHMOuterIndex	:= 1;
				tPerformanceRate := tonPerfomance.ET;

				eStep	:=E_CHM_FILECLOSE;
			ELSE
				bError 	:= TRUE;
				nErrorID	 := fbWriteCHMDataToXML.nErrorID;
				bSkipFLGFile	:= TRUE;

				eErrorState := eStep;

				eStep	:=E_CHM_FILECLOSE;
			END_IF

			bWriteCaseDataToXML := FALSE;
		END_IF

	E_CHM_FILECLOSE:

		(* close and release file for future use *)
		fbCloseFile(
			sNetId		:= '',
			hFile		:= hTarget,
			bExecute	:= TRUE,
			tTimeout	:= t#2s,
		);

		(* file close completed *)
		IF fbCloseFile.bBusy = FALSE THEN
			(* file close completed OK *)
			IF fbCloseFile.bError = FALSE THEN

				IF bSkipFLGFile OR NOT bIsValid THEN
					eStep	:=E_CHM_DONEGENERATOR;
				ELSE
					eStep	:=E_CHM_GENERATEFLG;
				END_IF
			(* file close error *)
			ELSE

				(* no previous error *)
				IF bError = FALSE THEN

					(* log error code and failure state *)
					bError := TRUE;
					nErrorID := fbCloseFile.nErrId;
					eErrorState := eStep;
				END_IF

				eStep	:=E_CHM_DONEGENERATOR;
			END_IF

			(* close off fbCloseFile *)
			fbCloseFile(bExecute := FALSE);
		END_IF

	E_CHM_GENERATEFLG:

		bCreatFLGFileExe := TRUE;

		IF	fbCreateFLGFile.bDone	 THEN

			IF NOT fbCreateFLGFile.bError THEN
				nSequenceNumber	:= nSequenceNumber+1;
			ELSE

				bError 	:= TRUE;
				nErrorID	 := fbCreateFLGFile.nErrorID;
				eErrorState := eStep;
			END_IF

			bCreatFLGFileExe := FALSE;

			eStep	:=E_CHM_DONEGENERATOR;
		END_IF

	E_CHM_DONEGENERATOR:

		MEMMOVE(ADR(stLastCaseHierarchyMessage), ADR(stCHMDataStruct), SIZEOF(stCHMDataStruct));
	
		bDone	:=  TRUE;
		bBusy	:=  FALSE;

		eStep	:=E_CHM_IDLEGENERATOR;
ELSE
	eStep	:=E_CHM_IDLEGENERATOR;
END_CASE

fbWriteCHMDataToXML(
	bExecute							:= bWriteCaseDataToXML,					(* set TRUE to write Case Produced file *)
	hTarget							:= hTarget,
	eMode								:= eCurrentXMLMode,
	nMaxPackItem						:= nMaxPackItem,
	nOuterIndex						:=nCHMOuterIndex,
	nCodingAndTrackingMode			:=nCodingAndTrackingMode,
	stAgregationData					:=stCHMDataStruct
);

rtrigFBDone(CLK:= fbWriteCHMDataToXML.bDone);

IF	rtrigFBDone.Q	THEN
	nLastImigeSize	:= fbWriteCHMDataToXML.nImageByte;
	MEMMOVE(ADR(aImigeSize[1]), ADR(aImigeSize), SIZEOF(aImigeSize)-SIZEOF(aImigeSize[1]));
	aImigeSize[0] := nLastImigeSize;
END_IF

fbCreateFLGFile(
	bExecute				:= bCreatFLGFileExe,					(* set TRUE to write Case Produced file *)
	sPath					:= sLocalCHMPath,			(* path for target file C:\CaseTrace*)
	sFLGFileName			:= sCHMFileName
);

END_FUNCTION_BLOCK

// ---- POUs/_Exclude/v3/FB_CHM_BiuldXMLImige_v3.TcPOU
FUNCTION_BLOCK FB_CHM_BiuldXMLImige_v3
VAR_INPUT
	bExecute					: BOOL;					(* set TRUE to write Case Produced file *)
	sCHMPathName			: STRING;
	eMode						: E_XML_WritingMode;
	nMaxPackItem				: UINT;
	nOuterIndex				: UINT;
	nCodingAndTrackingMode	: UINT;
END_VAR
VAR_IN_OUT
	hTarget					: UINT;
	stAgregationData	 			: ST_CHM_Data;		(* case data to be written to XML *)
END_VAR
VAR_OUTPUT
	bDone						: BOOL;					(* TRUE = XML file write complete *)
	bBusy						: BOOL;					(* TRUE = XML file write in progress *)
	bError						: BOOL;					(* TRUE = XML file write error *)
	nErrorID					: UDINT;				(* file write error code *)
	bVerifyError				: BOOL;					(* TRUE = XML file verification error *)
	nImageByte				: UDINT;
	nWriteImageSize			: UDINT;
END_VAR
VAR
	fbExecute					: R_TRIG;
	eState						: E_FILE_State;
	eErrorState					: E_FILE_State;

	ftrigOpen					: F_TRIG;
	ftrigWrite					: F_TRIG;
	ftrigClose					: F_TRIG;

	fbOpenFile					: FB_FileOpen;
	fbWriteFile					: FB_FileWrite;
	fbCloseFile					: FB_FileClose;

	hLastUsedTarget			: UINT;

	bGenerateImage			: BOOL;
	aXMLImage					: ARRAY[0..32767] OF BYTE;
	sString						: T_MaxString;
	nPackIndex				: UINT;

	nClose2Counter			: UINT;
	nChangeTargetCounter	: UINT;
	bReWrite					: BOOL;
END_VAR

(* rising edge of bExecute triggers new sequence *)
fbExecute(CLK := bExecute);

CASE eState OF

	(* waiting for trigger *)
	E_FILE_IDLE:

		(* rising edge of bExecute *)
		IF fbExecute.Q = TRUE THEN

			(* reset internal values *)
			bGenerateImage 	:= FALSE;
			MEMSET(ADR(aXMLImage), 16#00, SIZEOF(aXMLImage));
			nImageByte 		:= 0;
			nWriteImageSize 	:= 0;
			bReWrite			:= FALSE;

			(* update outputs *)
			bBusy 				:= TRUE;
			bDone 				:= FALSE;
			bError 				:= FALSE;
			nErrorID 			:= 0;
			bVerifyError		:= FALSE;

			eState := E_FILE_WRITE;

		(* bExecute has been reset *)
		ELSIF bExecute = FALSE THEN

			(* update outputs *)
			bBusy 				:= FALSE;
			bDone 				:= FALSE;
			bError 				:= FALSE;
			nErrorID 			:= 0;
			bVerifyError		:= FALSE;
		END_IF

	E_FILE_WRITE:

		IF NOT bGenerateImage THEN
			CASE eMode OF

				E_CS_HEADER:
					A_CaseHeaderGenerator();

				E_OUTER_HEADER:
					IF nCodingAndTrackingMode >= 7 THEN
						A_OuterHeaderContentGenerator();

						IF nCodingAndTrackingMode = 11 THEN
							FOR nPackIndex := 1 TO nMaxPackItem DO
								A_PackContentGenerator();
							END_FOR
						END_IF

						A_OuterEndPartGenerator();
					END_IF

				E_CS_ENDING:
					A_CaseEndPartGenerator();

			END_CASE

			bGenerateImage := TRUE;
		END_IF

		(* write data to open file *)
		fbWriteFile(
			sNetId		:= '',
			hFile		:= hTarget,
			pWriteBuff	:= ADR(aXMLImage),
			cbWriteLen	:= nImageByte,
			bExecute	:= TRUE,
			tTimeout	:= cTHREE_SECONDS
		);

		ftrigWrite(CLK:= fbWriteFile.bBusy) ;

		(* file write completed *)
		IF ftrigWrite.Q THEN

			(* file write completed OK *)
			IF fbWriteFile.bError = FALSE THEN

				(* log total bytes written *)
				nWriteImageSize := fbWriteFile.cbWrite;

				eState := E_FILE_DONE;
			(* file write error *)
			ELSE
				(* no previous error *)
				IF bReWrite = TRUE THEN

					(* log error code and failure state *)
					bError := TRUE;
					nErrorID := fbWriteFile.nErrId;
					eErrorState := eState;

					eState := E_FILE_DONE;
				ELSE
					eState := E_FILE_CLOSE;
				END_IF
			END_IF

			(* close off fbReadFile *)
			fbWriteFile(bExecute := FALSE);
		END_IF

	E_FILE_CLOSE:

	(* close and release file for future use *)
		fbCloseFile(
			sNetId		:= '',
			hFile		:= hTarget,
			bExecute	:= TRUE,
			tTimeout	:= t#1s,
		);

		ftrigClose(CLK:= fbCloseFile.bBusy) ;

		(* file close completed *)
		IF ftrigClose.Q THEN

			nClose2Counter := nClose2Counter + 1;

			eState := E_FILE_OPEN;

			(* close off fbCloseFile *)
			fbCloseFile(bExecute := FALSE);
		END_IF

	E_FILE_OPEN:

		fbOpenFile(
			sNetId		:= '',
			sPathName	:= sCHMPathName,
			nMode		:= FOPEN_MODEAPPEND OR FOPEN_MODEPLUS OR FOPEN_MODEBINARY,
			ePath		:= PATH_GENERIC,
			bExecute	:= TRUE,
			tTimeout	:= T#1s
		);

		ftrigOpen(CLK:= fbOpenFile.bBusy) ;

		(* file open completed *)
		IF  ftrigOpen.Q THEN

			(* file open completed OK *)
			IF fbOpenFile.bError = FALSE THEN

				IF fbOpenFile.hFile <> hTarget THEN
					(* log file handle for use by subsequent commands *)
					nChangeTargetCounter := nChangeTargetCounter+1;
					hLastUsedTarget	:= hTarget;
					hTarget := fbOpenFile.hFile;

				END_IF

				(* reset internal values *)
				bGenerateImage 	:= FALSE;
				MEMSET(ADR(aXMLImage), 16#00, SIZEOF(aXMLImage));
				nImageByte		:= 0;
				nWriteImageSize 	:= 0;
				bReWrite			:= TRUE;

				eState 				:= E_FILE_WRITE;

			(* file open error *)
			ELSE

				(* log error code and failure state *)
				bError := TRUE;
				nErrorID := fbOpenFile.nErrId;
				eErrorState := eState;

				(* abandon attempt to read file *)
				eState := E_FILE_DONE;
			END_IF

			(* close off fbOpenFile *)
			fbOpenFile(bExecute := FALSE);
		END_IF

	E_FILE_DONE:

		IF nImageByte <> nWriteImageSize THEN
			bVerifyError := TRUE;
		END_IF

		(* update outputs *)
		bBusy := FALSE;
		bDone := TRUE;

		eState := E_FILE_IDLE;
END_CASE

ACTION A_CaseEndPartGenerator:
	IF nCodingAndTrackingMode >= 7 THEN


				(* ItemList end*)
				sString := '$T$T$T$T</ItemList>$R$N';
				MEMMOVE(ADR(aXMLImage[nImageByte]), ADR(sString), LEN(sString));
				nImageByte := nImageByte + LEN(sString);

(***********CASE CONTENT END***********)
			(* Case Content END *)
			sString := '$T$T$T</Content>$R$N';
			MEMMOVE(ADR(aXMLImage[nImageByte]), ADR(sString), LEN(sString));
			nImageByte := nImageByte + LEN(sString);

	END_IF
			(* ProductionOrder *)
			sString := F_CONCAT3('$T$T$T<ProductionOrder>',stAgregationData.GenericHierarchy.CaseItem.ProductionOrder, '</ProductionOrder>$R$N');
			MEMMOVE(ADR(aXMLImage[nImageByte]), ADR(sString), LEN(sString));
			nImageByte := nImageByte + LEN(sString);

			(* LocalProductionOrder *)
			sString := F_CONCAT3('$T$T$T<LocalProductionOrder>',stAgregationData.GenericHierarchy.CaseItem.LocalProductionOrder, '</LocalProductionOrder>$R$N');
			MEMMOVE(ADR(aXMLImage[nImageByte]), ADR(sString), LEN(sString));
			nImageByte := nImageByte + LEN(sString);

			(* PITCode *)
			sString := F_CONCAT3('$T$T$T<PITCode>',stAgregationData.GenericHierarchy.CaseItem.PITCode, '</PITCode>$R$N');
			MEMMOVE(ADR(aXMLImage[nImageByte]), ADR(sString), LEN(sString));
			nImageByte := nImageByte + LEN(sString);

			(* BatchID *)
			sString := F_CONCAT3('$T$T$T<BatchID>',stAgregationData.GenericHierarchy.CaseItem.BatchID, '</BatchID>$R$N');
			MEMMOVE(ADR(aXMLImage[nImageByte]), ADR(sString), LEN(sString));
			nImageByte := nImageByte + LEN(sString);

			(* ProductionLine *)
			sString := F_CONCAT3('$T$T$T<ProductionLine>',stAgregationData.GenericHierarchy.CaseItem.ProductionLine, '</ProductionLine>$R$N');
			MEMMOVE(ADR(aXMLImage[nImageByte]), ADR(sString), LEN(sString));
			nImageByte := nImageByte + LEN(sString);


(***********Item CONTENT END***********)
		(* Item END *)
		sString := '$T$T</Item>$R$N';
		MEMMOVE(ADR(aXMLImage[nImageByte]), ADR(sString), LEN(sString));
		nImageByte := nImageByte + LEN(sString);

(***********GENERIC HIERARCHY CONTENT END***********)

	(* GenericHierarchy END *)
	sString := '$T</GenericHierarchy>$R$N';
	MEMMOVE(ADR(aXMLImage[nImageByte]), ADR(sString), LEN(sString));
	nImageByte := nImageByte + LEN(sString);

	(* Attributes *)
	sString := F_CONCAT3('$T<Attributes>', stAgregationData.Attributes, '</Attributes>$R$N');
	MEMMOVE(ADR(aXMLImage[nImageByte]), ADR(sString), LEN(sString));
	nImageByte := nImageByte + LEN(sString);

(* XPath leading tag  END*)
sString := '</GenericHierarchyList> $R$N';
MEMMOVE(ADR(aXMLImage[nImageByte]), ADR(sString), LEN(sString));
nImageByte := nImageByte + LEN(sString);
END_ACTION

ACTION A_CaseHeaderGenerator:
(* XML file version *)
(*sString := '<?xml version="1.0" encoding="utf-8"?>$R$N';
MEMMOVE(ADR(aXMLImage[nImageByte]), ADR(sString), LEN(sString));
nImageByte := nImageByte + LEN(sString);*)

(* XPath leading tag *)
sString := '<GenericHierarchyList xmlns:xsd="http://www.w3.org/2001/XMLSchema" xmlns:xsi="http://www.w3.org/2001/XMLSchema-instance"> $R$N';
MEMMOVE(ADR(aXMLImage[nImageByte]), ADR(sString), LEN(sString));
nImageByte := nImageByte + LEN(sString);

	(* MessageHeader *)
	sString := '$T<MessageHeader>$R$N';
	MEMMOVE(ADR(aXMLImage[nImageByte]), ADR(sString), LEN(sString));
	nImageByte := nImageByte + LEN(sString);

(***********MESSAGE HEADER CONTENT***********)

		(*(* CreationDate *)
		sString := F_CONCAT3('$T$T<CreationDate>',stAgregationData.MessageHeader.CreationDate, '</CreationDate>$R$N');
		MEMMOVE(ADR(aXMLImage[nImageByte]), ADR(sString), LEN(sString));
		nImageByte := nImageByte + LEN(sString);
	
		(* CreationTime *)
		sString := F_CONCAT3('$T$T<CreationTime>',stAgregationData.MessageHeader.CreationTime, '</CreationTime>$R$N');
		MEMMOVE(ADR(aXMLImage[nImageByte]), ADR(sString), LEN(sString));
		nImageByte := nImageByte + LEN(sString);*)

		(* ReferenceID *)
		sString := F_CONCAT3('$T$T<ReferenceID>',stAgregationData.MessageHeader.ReferenceID, '</ReferenceID>$R$N');
		MEMMOVE(ADR(aXMLImage[nImageByte]), ADR(sString), LEN(sString));
		nImageByte := nImageByte + LEN(sString);

		(* CreationTimeLocalUTC *)
		sString := F_CONCAT3('$T$T<CreationTimeLocalUTC>',stAgregationData.MessageHeader.CreationTimeLocalUTC, '</CreationTimeLocalUTC>$R$N');
		MEMMOVE(ADR(aXMLImage[nImageByte]), ADR(sString), LEN(sString));
		nImageByte := nImageByte + LEN(sString);

		(* MessageType *)
		sString := F_CONCAT3('$T$T<MessageType>',stAgregationData.MessageHeader.MessageType, '</MessageType>$R$N');
		MEMMOVE(ADR(aXMLImage[nImageByte]), ADR(sString), LEN(sString));
		nImageByte := nImageByte + LEN(sString);

		(* SenderSystem *)
		sString := F_CONCAT3('$T$T<SenderSystem>',stAgregationData.MessageHeader.SenderSystem, '</SenderSystem>$R$N');
		MEMMOVE(ADR(aXMLImage[nImageByte]), ADR(sString), LEN(sString));
		nImageByte := nImageByte + LEN(sString);

		(* ReceiverSystem *)
		sString := F_CONCAT3('$T$T<ReceiverSystem>',stAgregationData.MessageHeader.ReceiverSystem, '</ReceiverSystem>$R$N');
		MEMMOVE(ADR(aXMLImage[nImageByte]), ADR(sString), LEN(sString));
		nImageByte := nImageByte + LEN(sString);

(***********MESSAGE HEADER CONTENT END***********)

	(* MessageHeader END *)
	sString := '$T</MessageHeader>$R$N';
	MEMMOVE(ADR(aXMLImage[nImageByte]), ADR(sString), LEN(sString));
	nImageByte := nImageByte + LEN(sString);

	(* Factory*)
	sString := F_CONCAT3('$T<Factory>', stAgregationData.Factory, '</Factory>$R$N');
	MEMMOVE(ADR(aXMLImage[nImageByte]), ADR(sString), LEN(sString));
	nImageByte := nImageByte + LEN(sString);

	(* GenericHierarchy *)
	sString := '$T<GenericHierarchy>$R$N';
	MEMMOVE(ADR(aXMLImage[nImageByte]), ADR(sString), LEN(sString));
	nImageByte := nImageByte + LEN(sString);

(***********GENERIC HIERARCHY CONTENT***********)

		(* HierarchyType *)
		sString := F_CONCAT3('$T$T<HierarchyType>',stAgregationData.GenericHierarchy.HierarchyType, '</HierarchyType>$R$N');
		MEMMOVE(ADR(aXMLImage[nImageByte]), ADR(sString), LEN(sString));
		nImageByte := nImageByte + LEN(sString);

		(* PerformedAction *)
		sString := F_CONCAT3('$T$T<ACTION>',stAgregationData.GenericHierarchy.PerformedAction, '</ACTION>$R$N');
		MEMMOVE(ADR(aXMLImage[nImageByte]), ADR(sString), LEN(sString));
		nImageByte := nImageByte + LEN(sString);

		(* TrackingLevels *)
		sString := F_CONCAT3('$T$T<TrackingLevels>',stAgregationData.GenericHierarchy.TrackingLevels, '</TrackingLevels>$R$N');
		MEMMOVE(ADR(aXMLImage[nImageByte]), ADR(sString), LEN(sString));
		nImageByte := nImageByte + LEN(sString);

		(* TrackingIndicator *)
		sString := F_CONCAT3('$T$T<TrackingIndicator>',stAgregationData.GenericHierarchy.TrackingIndicator, '</TrackingIndicator>$R$N');
		MEMMOVE(ADR(aXMLImage[nImageByte]), ADR(sString), LEN(sString));
		nImageByte := nImageByte + LEN(sString);

		(* Item Type *)
		sString := '$T$T<Item Type="CS">$R$N';
		MEMMOVE(ADR(aXMLImage[nImageByte]), ADR(sString), LEN(sString));
		nImageByte := nImageByte + LEN(sString);

(***********Item Type CONTENT***********)
			(* Identity*)
			sString := '$T$T$T<Identity>$R$N';
			MEMMOVE(ADR(aXMLImage[nImageByte]), ADR(sString), LEN(sString));
			nImageByte := nImageByte + LEN(sString);

(***********Identity CONTENT***********)
					(* SKU *)
					sString := F_CONCAT3('$T$T$T$T<SKU>',stAgregationData.GenericHierarchy.CaseItem.Identity.SKU, '</SKU>$R$N');
					MEMMOVE(ADR(aXMLImage[nImageByte]), ADR(sString), LEN(sString));
					nImageByte := nImageByte + LEN(sString);

					(* GTIN *)
					sString := F_CONCAT3('$T$T$T$T<GTIN>',stAgregationData.GenericHierarchy.CaseItem.Identity.GTIN, '</GTIN>$R$N');
					MEMMOVE(ADR(aXMLImage[nImageByte]), ADR(sString), LEN(sString));
					nImageByte := nImageByte + LEN(sString);

					(* ID *)
					sString := F_CONCAT3('$T$T$T$T<ID>',stAgregationData.GenericHierarchy.CaseItem.Identity.ID, '</ID>$R$N');
					MEMMOVE(ADR(aXMLImage[nImageByte]), ADR(sString), LEN(sString));
					nImageByte := nImageByte + LEN(sString);

					(* ReadQuality *)
					sString := F_CONCAT3('$T$T$T$T<ReadQuality>',stAgregationData.GenericHierarchy.CaseItem.Identity.ReadQuality, '</ReadQuality>$R$N');
					MEMMOVE(ADR(aXMLImage[nImageByte]), ADR(sString), LEN(sString));
					nImageByte := nImageByte + LEN(sString);

(***********Identity CONTENT END***********)

			(* Identity END *)
			sString := '$T$T$T</Identity>$R$N';
			MEMMOVE(ADR(aXMLImage[nImageByte]), ADR(sString), LEN(sString));
			nImageByte := nImageByte + LEN(sString);

			(* ItemState *)
			sString := F_CONCAT3('$T$T$T<ItemState>',stAgregationData.GenericHierarchy.CaseItem.ItemState, '</ItemState>$R$N');
			MEMMOVE(ADR(aXMLImage[nImageByte]), ADR(sString), LEN(sString));
			nImageByte := nImageByte + LEN(sString);

			(* RejectReason *)
			sString := '$T$T$T<RejectReason>$R$N';
			MEMMOVE(ADR(aXMLImage[nImageByte]), ADR(sString), LEN(sString));
			nImageByte := nImageByte + LEN(sString);

				sString := F_CONCAT3('$T$T$T$T<Reason>',stAgregationData.GenericHierarchy.CaseItem.RejectReason, '</Reason>$R$N');
				MEMMOVE(ADR(aXMLImage[nImageByte]), ADR(sString), LEN(sString));
				nImageByte := nImageByte + LEN(sString);

			sString := '$T$T$T</RejectReason>$R$N';
			MEMMOVE(ADR(aXMLImage[nImageByte]), ADR(sString), LEN(sString));
			nImageByte := nImageByte + LEN(sString);

			(*logs *)
			sString := '$T$T$T<logs>$R$N';
			MEMMOVE(ADR(aXMLImage[nImageByte]), ADR(sString), LEN(sString));
			nImageByte := nImageByte + LEN(sString);

				(* TimeStamp *)
				sString := F_CONCAT3('$T$T$T$T<TimeStamp Topic="Aggregation">',stAgregationData.GenericHierarchy.CaseItem.TimeStamp, '</TimeStamp>$R$N');
				MEMMOVE(ADR(aXMLImage[nImageByte]), ADR(sString), LEN(sString));
				nImageByte := nImageByte + LEN(sString);

			(* logs END *)
			sString := '$T$T$T</logs>$R$N';
			MEMMOVE(ADR(aXMLImage[nImageByte]), ADR(sString), LEN(sString));
			nImageByte := nImageByte + LEN(sString);

			(* NoRead *)
			sString := F_CONCAT3('$T$T$T<NoRead>',stAgregationData.GenericHierarchy.CaseItem.NoRead, '</NoRead>$R$N');
			MEMMOVE(ADR(aXMLImage[nImageByte]), ADR(sString), LEN(sString));
			nImageByte := nImageByte + LEN(sString);

(***********CONTENT***********)
	IF nCodingAndTrackingMode >= 7 THEN

			(* Case Content *)
			sString := '$T$T$T<Content>$R$N';
			MEMMOVE(ADR(aXMLImage[nImageByte]), ADR(sString), LEN(sString));
			nImageByte := nImageByte + LEN(sString);

				(* Case DefaultIdentity*)
				sString := '$T$T$T$T<DefaultIdentity>$R$N';
				MEMMOVE(ADR(aXMLImage[nImageByte]), ADR(sString), LEN(sString));
				nImageByte := nImageByte + LEN(sString);

						(* SKU *)
						sString := F_CONCAT3('$T$T$T$T$T<SKU>',stAgregationData.GenericHierarchy.CaseItem.Content.DefaultIdentity.SKU, '</SKU>$R$N');
						MEMMOVE(ADR(aXMLImage[nImageByte]), ADR(sString), LEN(sString));
						nImageByte := nImageByte + LEN(sString);

						(* GTIN *)
						sString := F_CONCAT3('$T$T$T$T$T<GTIN>',stAgregationData.GenericHierarchy.CaseItem.Content.DefaultIdentity.GTIN, '</GTIN>$R$N');
						MEMMOVE(ADR(aXMLImage[nImageByte]), ADR(sString), LEN(sString));
						nImageByte := nImageByte + LEN(sString);

						(* ProductionOrder *)
						sString := F_CONCAT3('$T$T$T$T$T<ProductionOrder>',stAgregationData.GenericHierarchy.CaseItem.Content.DefaultIdentity.ProductionOrder, '</ProductionOrder>$R$N');
						MEMMOVE(ADR(aXMLImage[nImageByte]), ADR(sString), LEN(sString));
						nImageByte := nImageByte + LEN(sString);

						(* LocalProductionOrder *)
						sString := F_CONCAT3('$T$T$T$T$T<LocalProductionOrder>',stAgregationData.GenericHierarchy.CaseItem.Content.DefaultIdentity.LocalProductionOrder, '</LocalProductionOrder>$R$N');
						MEMMOVE(ADR(aXMLImage[nImageByte]), ADR(sString), LEN(sString));
						nImageByte := nImageByte + LEN(sString);

						(* PITCode *)
						sString := F_CONCAT3('$T$T$T$T$T<PITCode>',stAgregationData.GenericHierarchy.CaseItem.Content.DefaultIdentity.PITCode, '</PITCode>$R$N');
						MEMMOVE(ADR(aXMLImage[nImageByte]), ADR(sString), LEN(sString));
						nImageByte := nImageByte + LEN(sString);

						(* BatchID *)
						sString := F_CONCAT3('$T$T$T$T$T<BatchID>',stAgregationData.GenericHierarchy.CaseItem.Content.DefaultIdentity.BatchID, '</BatchID>$R$N');
						MEMMOVE(ADR(aXMLImage[nImageByte]), ADR(sString), LEN(sString));
						nImageByte := nImageByte + LEN(sString);

						(* ProductionLine *)
						sString := F_CONCAT3('$T$T$T$T$T<ProductionLine>',stAgregationData.GenericHierarchy.CaseItem.Content.DefaultIdentity.ProductionLine, '</ProductionLine>$R$N');
						MEMMOVE(ADR(aXMLImage[nImageByte]), ADR(sString), LEN(sString));
						nImageByte := nImageByte + LEN(sString);

				(* Case DefaultIdentity END*)
				sString := '$T$T$T$T</DefaultIdentity>$R$N';
				MEMMOVE(ADR(aXMLImage[nImageByte]), ADR(sString), LEN(sString));
				nImageByte := nImageByte + LEN(sString);

				(* ExpectedItemCount *)
				sString := F_CONCAT3('$T$T$T$T<ExpectedItemCount>',stAgregationData.GenericHierarchy.CaseItem.Content.ExpectedItemCount, '</ExpectedItemCount>$R$N');
				MEMMOVE(ADR(aXMLImage[nImageByte]), ADR(sString), LEN(sString));
				nImageByte := nImageByte + LEN(sString);

				(* ItemReadRate *)
				sString := F_CONCAT3('$T$T$T$T<ItemReadRate>',stAgregationData.GenericHierarchy.CaseItem.Content.ItemReadRate, '</ItemReadRate>$R$N');
				MEMMOVE(ADR(aXMLImage[nImageByte]), ADR(sString), LEN(sString));
				nImageByte := nImageByte + LEN(sString);

				(* ItemList*)
				sString := '$T$T$T$T<ItemList>$R$N';
				MEMMOVE(ADR(aXMLImage[nImageByte]), ADR(sString), LEN(sString));
				nImageByte := nImageByte + LEN(sString);
	END_IF
END_ACTION

ACTION A_OuterEndPartGenerator:
(*
    </ItemList> 
                        </Content> 
                    </Item> 

*)
						IF nCodingAndTrackingMode = 11 THEN
								(* ItemList end*)
								sString := '$T$T$T$T$T$T$T</ItemList>$R$N';
								MEMMOVE(ADR(aXMLImage[nImageByte]), ADR(sString), LEN(sString));
								nImageByte := nImageByte + LEN(sString);
	(***********CASE CONTENT END***********)
							(* Outer Content END *)
							sString := '$T$T$T$T$T$T</Content>$R$N';
							MEMMOVE(ADR(aXMLImage[nImageByte]), ADR(sString), LEN(sString));
							nImageByte := nImageByte + LEN(sString);
						END_IF

								(* Item Type END *)
								sString := '$T$T$T$T$T</Item>$R$N';
							MEMMOVE(ADR(aXMLImage[nImageByte]), ADR(sString), LEN(sString));
							nImageByte := nImageByte + LEN(sString);
END_ACTION

ACTION A_OuterHeaderContentGenerator:
(*
                  <Item Type="OUT"> 
                        <Identity> 
                         	   <ID>55128CY203644964300</ID> 
                        	    <ReadQuality>100</ReadQuality> 
                        </Identity> 
                        <ItemState>Verified</ItemState> 
                        <RejectReason /> 
                        <logs> 
                   		        <TimeStamp Topic="Aggregation">2018-03-22T20:46:01.5229666+01:00</TimeStamp> 
                        </logs> 
                        <NoRead>false</NoRead> 
                        <Content> 
                           	 <DefaultIdentity> 
                      	     	     <SKU>10045622</SKU> 
                        	   	     <GTIN>00000087295993</GTIN> 
                        		        <ProductionOrder>2523549</ProductionOrder> 
                         		       <LocalProductionOrder>2523549</LocalProductionOrder> 
                           		     <PITCode>3</PITCode> 
                          		      <BatchID>55122018</BatchID> 
                        		        <ProductionLine>12</ProductionLine> 
                       	     </DefaultIdentity> 
                      	      <ExpectedItemCount>10</ExpectedItemCount> 
                       	     <ItemReadRate>100</ItemReadRate> 
                       	     <ItemList> 

*)


					(* Item Type *)
					sString := '$T$T$T$T$T<Item Type="OUT">$R$N';
					MEMMOVE(ADR(aXMLImage[nImageByte]), ADR(sString), LEN(sString));
					nImageByte := nImageByte + LEN(sString);

						(* Identity *)
						sString := '$T$T$T$T$T$T<Identity>$R$N';
						MEMMOVE(ADR(aXMLImage[nImageByte]), ADR(sString), LEN(sString));
						nImageByte := nImageByte + LEN(sString);

							(* ID *)
							sString := F_CONCAT3('$T$T$T$T$T$T$T<ID><![CDATA[',stAgregationData.GenericHierarchy.CaseItem.Content.arrOuterItem[nOuterIndex].Identity.ID, ']]></ID>$R$N');
							MEMMOVE(ADR(aXMLImage[nImageByte]), ADR(sString), LEN(sString));
							nImageByte := nImageByte + LEN(sString);

							(* ReadQuality *)
							sString := F_CONCAT3('$T$T$T$T$T$T$T<ReadQuality>',stAgregationData.GenericHierarchy.CaseItem.Content.arrOuterItem[nOuterIndex].Identity.ReadQuality, '</ReadQuality>$R$N');
							MEMMOVE(ADR(aXMLImage[nImageByte]), ADR(sString), LEN(sString));
							nImageByte := nImageByte + LEN(sString);

						(* Identity END *)
						sString := '$T$T$T$T$T$T</Identity>$R$N';
						MEMMOVE(ADR(aXMLImage[nImageByte]), ADR(sString), LEN(sString));
						nImageByte := nImageByte + LEN(sString);


